LIN {X 0,Y 412.15,Z 242.134,A -85,B 0,C 180,E1 -10569.119,E2 -10569.119} C_VEL
LIN {X 0,Y 411.731,Z 238.226,A -85,B 0,C 180,E1 -10571.737,E2 -10571.737} C_VEL
LIN {X 0,Y 411.199,Z 234.89,A -85,B 0,C 180,E1 -10574.123,E2 -10574.123} C_VEL
LIN {X 0,Y 411.182,Z 234.895,A -85,B 0,C 180,E1 -10577.304,E2 -10577.304} C_VEL
LIN {X 0,Y 411.215,Z 234.89,A -85,B 0,C 180,E1 -10580.776,E2 -10580.776} C_VEL
LIN {X 0,Y 411.198,Z 234.894,A -85,B 0,C 180,E1 -10584.471,E2 -10584.471} C_VEL
LIN {X 0,Y 411.208,Z 234.889,A -85,B 0,C 180,E1 -10586.873,E2 -10586.873} C_VEL
LIN {X 0,Y 411.212,Z 234.891,A -85,B 0,C 180,E1 -10590.65,E2 -10590.65} C_VEL
LIN {X 0,Y 411.195,Z 234.89,A -85,B 0,C 180,E1 -10593.616,E2 -10593.616} C_VEL
LIN {X 0,Y 411.196,Z 234.89,A -85,B 0,C 180,E1 -10596.852,E2 -10596.852} C_VEL
LIN {X 0,Y 411.216,Z 234.887,A -85,B 0,C 180,E1 -10600.051,E2 -10600.051} C_VEL
LIN {X 0,Y 411.264,Z 234.879,A -85,B 0,C 180,E1 -10603.131,E2 -10603.131} C_VEL
LIN {X 0,Y 411.307,Z 234.877,A -85,B 0,C 180,E1 -10606.896,E2 -10606.896} C_VEL
LIN {X 0,Y 411.29,Z 234.876,A -85,B 0,C 180,E1 -10610.161,E2 -10610.161} C_VEL
LIN {X 0,Y 411.394,Z 234.865,A -85,B 0,C 180,E1 -10613.132,E2 -10613.132} C_VEL
LIN {X 0,Y 411.303,Z 234.878,A -85,B 0,C 180,E1 -10615.099,E2 -10615.099} C_VEL
LIN {X 0,Y 411.513,Z 234.851,A -85,B 0,C 180,E1 -10618.043,E2 -10618.043} C_VEL
LIN {X 0,Y 411.635,Z 234.837,A -85,B 0,C 180,E1 -10620,E2 -10620} C_VEL
LIN {X 0,Y 411.449,Z 234.859,A -85,B 0,C 180,E1 -10622.937,E2 -10622.937} C_VEL
LIN {X 0,Y 411.448,Z 234.857,A -85,B 0,C 180,E1 -10626.672,E2 -10626.672} C_VEL
LIN {X 0,Y 411.294,Z 234.88,A -85,B 0,C 180,E1 -10629.839,E2 -10629.839} C_VEL
LIN {X 0,Y 411.307,Z 234.877,A -85,B 0,C 180,E1 -10633.104,E2 -10633.104} C_VEL
LIN {X 0,Y 411.259,Z 234.881,A -85,B 0,C 180,E1 -10636.889,E2 -10636.889} C_VEL
LIN {X 0,Y 411.232,Z 234.884,A -85,B 0,C 180,E1 -10639.987,E2 -10639.987} C_VEL
LIN {X 0,Y 411.197,Z 234.889,A -85,B 0,C 180,E1 -10643.148,E2 -10643.148} C_VEL
LIN {X 0,Y 411.238,Z 234.884,A -85,B 0,C 180,E1 -10646.381,E2 -10646.381} C_VEL
LIN {X 0,Y 411.202,Z 234.888,A -85,B 0,C 180,E1 -10649.713,E2 -10649.713} C_VEL
LIN {X 0,Y 411.208,Z 234.887,A -85,B 0,C 180,E1 -10653.156,E2 -10653.156} C_VEL
LIN {X 0,Y 411.194,Z 234.889,A -85,B 0,C 180,E1 -10656.553,E2 -10656.553} C_VEL
LIN {X 0,Y 411.179,Z 234.89,A -85,B 0,C 180,E1 -10659.722,E2 -10659.722} C_VEL
LIN {X 0,Y 411.166,Z 234.895,A -85,B 0,C 180,E1 -10663.135,E2 -10663.135} C_VEL
LIN {X 0,Y 411.169,Z 234.895,A -85,B 0,C 180,E1 -10665.881,E2 -10665.881} C_VEL
LIN {X 0,Y 411.159,Z 234.898,A -85,B 0,C 180,E1 -10668.773,E2 -10668.773} C_VEL
LIN {X 0,Y 411.159,Z 234.896,A -85,B 0,C 180,E1 -10669.493,E2 -10669.493} C_VEL
LIN {X 0,Y 411.277,Z 236.124,A -85,B 0,C 180,E1 -10670.782,E2 -10670.782} C_VEL
LIN {X 0,Y 411.294,Z 239.248,A -85,B 0,C 180,E1 -10673.429,E2 -10673.429} C_VEL
LIN {X 0,Y 411.162,Z 241.979,A -85,B 0,C 180,E1 -10675.662,E2 -10675.662} C_VEL
LIN {X 0,Y 410.925,Z 246.363,A -85,B 0,C 180,E1 -10679.13,E2 -10679.13} C_VEL
LIN {X 0,Y 410.666,Z 250.766,A -85,B 0,C 180,E1 -10682.479,E2 -10682.479} C_VEL
LIN {X 0,Y 410.562,Z 255.215,A -85,B 0,C 180,E1 -10685.743,E2 -10685.743} C_VEL
LIN {X 0,Y 410.436,Z 259.421,A -85,B 0,C 180,E1 -10688.752,E2 -10688.752} C_VEL
LIN {X 0,Y 414.52,Z 274.317,A -85,B 0,C 180,E1 -10689.4,E2 -10689.4} C_VEL
LIN {X 0,Y 417.537,Z 287.727,A -85,B 0,C 180,E1 -10690.136,E2 -10690.136} C_VEL
LIN {X 0,Y 417.676,Z 291.393,A -85,B 0,C 180,E1 -10690.335,E2 -10690.335} C_VEL
LIN {X 0,Y 416.878,Z 304.123,A -85,B 0,C 180,E1 -10691.091,E2 -10691.091} C_VEL
LIN {X 0,Y 415.949,Z 316.643,A -85,B 0,C 180,E1 -10692.04,E2 -10692.04} C_VEL
LIN {X 0,Y 414.909,Z 328.342,A -85,B 0,C 180,E1 -10693.138,E2 -10693.138} C_VEL
LIN {X 0,Y 413.823,Z 340.015,A -85,B 0,C 180,E1 -10694.485,E2 -10694.485} C_VEL
LIN {X 0,Y 412.756,Z 350.606,A -85,B 0,C 180,E1 -10695.983,E2 -10695.983} C_VEL
LIN {X 0,Y 412.086,Z 359.036,A -85,B 0,C 180,E1 -10697.441,E2 -10697.441} C_VEL
LIN {X 0,Y 411.263,Z 367.277,A -85,B 0,C 180,E1 -10699.165,E2 -10699.165} C_VEL
LIN {X 0,Y 410.811,Z 373.015,A -85,B 0,C 180,E1 -10700.647,E2 -10700.647} C_VEL
LIN {X 0,Y 410.452,Z 377.734,A -85,B 0,C 180,E1 -10702.127,E2 -10702.127} C_VEL
LIN {X 0,Y 410.322,Z 381.154,A -85,B 0,C 180,E1 -10703.428,E2 -10703.428} C_VEL
LIN {X 0,Y 410.101,Z 384.499,A -85,B 0,C 180,E1 -10705.085,E2 -10705.085} C_VEL
LIN {X 0,Y 409.972,Z 387.2,A -85,B 0,C 180,E1 -10707.052,E2 -10707.052} C_VEL
LIN {X 0,Y 409.918,Z 388.555,A -85,B 0,C 180,E1 -10709.018,E2 -10709.018} C_VEL
LIN {X 0,Y 409.918,Z 388.591,A -85,B 0,C 180,E1 -10710.982,E2 -10710.982} C_VEL
LIN {X 0,Y 409.971,Z 387.304,A -85,B 0,C 180,E1 -10712.948,E2 -10712.948} C_VEL
LIN {X 0,Y 410.095,Z 384.665,A -85,B 0,C 180,E1 -10714.916,E2 -10714.916} C_VEL
LIN {X 0,Y 410.321,Z 380.607,A -85,B 0,C 180,E1 -10716.886,E2 -10716.886} C_VEL
LIN {X 0,Y 410.591,Z 375.976,A -85,B 0,C 180,E1 -10718.557,E2 -10718.557} C_VEL
LIN {X 0,Y 410.123,Z 373.603,A -85,B 0,C 180,E1 -10719.305,E2 -10719.305} C_VEL
LIN {X 0,Y 407.665,Z 369.385,A -85,B 0,C 180,E1 -10720.516,E2 -10720.516} C_VEL
LIN {X 0,Y 405.273,Z 364.741,A -85,B 0,C 180,E1 -10721.704,E2 -10721.704} C_VEL
LIN {X 0,Y 404.912,Z 361.52,A -85,B 0,C 180,E1 -10722.406,E2 -10722.406} C_VEL
LIN {X 0,Y 405.639,Z 352.68,A -85,B 0,C 180,E1 -10724.038,E2 -10724.038} C_VEL
LIN {X 0,Y 406.716,Z 342.744,A -85,B 0,C 180,E1 -10725.536,E2 -10725.536} C_VEL
LIN {X 0,Y 407.811,Z 331.683,A -85,B 0,C 180,E1 -10726.907,E2 -10726.907} C_VEL
LIN {X 0,Y 409.011,Z 319.268,A -85,B 0,C 180,E1 -10728.146,E2 -10728.146} C_VEL
LIN {X 0,Y 409.999,Z 307.073,A -85,B 0,C 180,E1 -10729.129,E2 -10729.129} C_VEL
LIN {X 0,Y 410.827,Z 294.562,A -85,B 0,C 180,E1 -10729.931,E2 -10729.931} C_VEL
LIN {X 0,Y 411.06,Z 290.348,A -85,B 0,C 180,E1 -10730.162,E2 -10730.162} C_VEL
LIN {X 0,Y 408.229,Z 277.162,A -85,B 0,C 180,E1 -10730.932,E2 -10730.932} C_VEL
LIN {X 0,Y 404.44,Z 263.529,A -85,B 0,C 180,E1 -10731.585,E2 -10731.585} C_VEL
LIN {X 0,Y 403.377,Z 259.517,A -85,B 0,C 180,E1 -10731.764,E2 -10731.764} C_VEL
LIN {X 0,Y 403.543,Z 254.954,A -85,B 0,C 180,E1 -10735.093,E2 -10735.093} C_VEL
LIN {X 0,Y 403.639,Z 251.022,A -85,B 0,C 180,E1 -10738.042,E2 -10738.042} C_VEL
LIN {X 0,Y 403.826,Z 248.062,A -85,B 0,C 180,E1 -10740.312,E2 -10740.312} C_VEL
LIN {X 0,Y 404.083,Z 243.693,A -85,B 0,C 180,E1 -10743.818,E2 -10743.818} C_VEL
LIN {X 0,Y 404.248,Z 239.971,A -85,B 0,C 180,E1 -10746.896,E2 -10746.896} C_VEL
LIN {X 0,Y 404.171,Z 236.332,A -85,B 0,C 180,E1 -10750.045,E2 -10750.045} C_VEL
LIN {X 0,Y 404.119,Z 235.775,A -85,B 0,C 180,E1 -10751.599,E2 -10751.599} C_VEL
LIN {X 0,Y 404.148,Z 235.771,A -85,B 0,C 180,E1 -10754.522,E2 -10754.522} C_VEL
LIN {X 0,Y 404.127,Z 235.772,A -85,B 0,C 180,E1 -10757.294,E2 -10757.294} C_VEL
LIN {X 0,Y 404.134,Z 235.77,A -85,B 0,C 180,E1 -10759.951,E2 -10759.951} C_VEL
LIN {X 0,Y 404.138,Z 235.77,A -85,B 0,C 180,E1 -10763.125,E2 -10763.125} C_VEL
LIN {X 0,Y 404.147,Z 235.77,A -85,B 0,C 180,E1 -10766.188,E2 -10766.188} C_VEL
LIN {X 0,Y 404.148,Z 235.768,A -85,B 0,C 180,E1 -10769.715,E2 -10769.715} C_VEL
LIN {X 0,Y 404.198,Z 235.761,A -85,B 0,C 180,E1 -10773.123,E2 -10773.123} C_VEL
LIN {X 0,Y 404.177,Z 235.76,A -85,B 0,C 180,E1 -10775.334,E2 -10775.334} C_VEL
LIN {X 0,Y 404.141,Z 235.768,A -85,B 0,C 180,E1 -10778.581,E2 -10778.581} C_VEL
LIN {X 0,Y 404.211,Z 235.759,A -85,B 0,C 180,E1 -10781.762,E2 -10781.762} C_VEL
LIN {X 0,Y 404.209,Z 235.759,A -85,B 0,C 180,E1 -10784.882,E2 -10784.882} C_VEL
LIN {X 0,Y 404.259,Z 235.753,A -85,B 0,C 180,E1 -10787.958,E2 -10787.958} C_VEL
LIN {X 0,Y 404.269,Z 235.751,A -85,B 0,C 180,E1 -10790.998,E2 -10790.998} C_VEL
LIN {X 0,Y 404.417,Z 235.733,A -85,B 0,C 180,E1 -10794.015,E2 -10794.015} C_VEL
LIN {X 0,Y 404.48,Z 235.725,A -85,B 0,C 180,E1 -10798.008,E2 -10798.008} C_VEL
LIN {X 0,Y 404.42,Z 235.733,A -85,B 0,C 180,E1 -10800.996,E2 -10800.996} C_VEL
LIN {X 0,Y 404.418,Z 235.733,A -85,B 0,C 180,E1 -10802.988,E2 -10802.988} C_VEL
LIN {X 0,Y 404.384,Z 235.738,A -85,B 0,C 180,E1 -10805.985,E2 -10805.985} C_VEL
LIN {X 0,Y 404.267,Z 235.752,A -85,B 0,C 180,E1 -10809.001,E2 -10809.001} C_VEL
LIN {X 0,Y 404.259,Z 235.752,A -85,B 0,C 180,E1 -10812.041,E2 -10812.041} C_VEL
LIN {X 0,Y 404.21,Z 235.761,A -85,B 0,C 180,E1 -10815.118,E2 -10815.118} C_VEL
LIN {X 0,Y 404.206,Z 235.761,A -85,B 0,C 180,E1 -10818.238,E2 -10818.238} C_VEL
LIN {X 0,Y 404.141,Z 235.77,A -85,B 0,C 180,E1 -10821.419,E2 -10821.419} C_VEL
LIN {X 0,Y 404.163,Z 235.764,A -85,B 0,C 180,E1 -10824.667,E2 -10824.667} C_VEL
LIN {X 0,Y 404.118,Z 235.771,A -85,B 0,C 180,E1 -10828.005,E2 -10828.005} C_VEL
LIN {X 0,Y 404.146,Z 235.768,A -85,B 0,C 180,E1 -10830.285,E2 -10830.285} C_VEL
LIN {X 0,Y 404.147,Z 235.769,A -85,B 0,C 180,E1 -10833.812,E2 -10833.812} C_VEL
LIN {X 0,Y 404.137,Z 235.772,A -85,B 0,C 180,E1 -10836.875,E2 -10836.875} C_VEL
LIN {X 0,Y 404.149,Z 235.769,A -85,B 0,C 180,E1 -10840.08,E2 -10840.08} C_VEL
LIN {X 0,Y 404.155,Z 235.772,A -85,B 0,C 180,E1 -10843.084,E2 -10843.084} C_VEL
LIN {X 0,Y 404.162,Z 235.921,A -85,B 0,C 180,E1 -10845.71,E2 -10845.71} C_VEL
LIN {X 0,Y 404.829,Z 240.125,A -85,B 0,C 180,E1 -10848.723,E2 -10848.723} C_VEL
LIN {X 0,Y 405.166,Z 244.034,A -85,B 0,C 180,E1 -10851.358,E2 -10851.358} C_VEL
LIN {X 0,Y 404.996,Z 247.953,A -85,B 0,C 180,E1 -10853.842,E2 -10853.842} C_VEL
LIN {X 0,Y 404.579,Z 253.839,A -85,B 0,C 180,E1 -10857.418,E2 -10857.418} C_VEL
LIN {X 0,Y 404.232,Z 259.74,A -85,B 0,C 180,E1 -10860.869,E2 -10860.869} C_VEL
LIN {X 0,Y 404.002,Z 263.62,A -85,B 0,C 180,E1 -10863.109,E2 -10863.109} C_VEL
LIN {X 0,Y 403.608,Z 269.448,A -85,B 0,C 180,E1 -10866.391,E2 -10866.391} C_VEL
LIN {X 0,Y 403.506,Z 272.965,A -85,B 0,C 180,E1 -10868.3,E2 -10868.3} C_VEL
LIN {X 0,Y 407.021,Z 287.509,A -85,B 0,C 180,E1 -10868.898,E2 -10868.898} C_VEL
LIN {X 0,Y 409.374,Z 299.361,A -85,B 0,C 180,E1 -10869.512,E2 -10869.512} C_VEL
LIN {X 0,Y 410.559,Z 307.1,A -85,B 0,C 180,E1 -10869.979,E2 -10869.979} C_VEL
LIN {X 0,Y 409.743,Z 319.944,A -85,B 0,C 180,E1 -10870.769,E2 -10870.769} C_VEL
LIN {X 0,Y 408.695,Z 332.088,A -85,B 0,C 180,E1 -10871.71,E2 -10871.71} C_VEL
LIN {X 0,Y 407.583,Z 343.741,A -85,B 0,C 180,E1 -10872.825,E2 -10872.825} C_VEL
LIN {X 0,Y 406.637,Z 353.442,A -85,B 0,C 180,E1 -10873.947,E2 -10873.947} C_VEL
LIN {X 0,Y 405.605,Z 364.193,A -85,B 0,C 180,E1 -10875.449,E2 -10875.449} C_VEL
LIN {X 0,Y 404.793,Z 373.072,A -85,B 0,C 180,E1 -10876.955,E2 -10876.955} C_VEL
LIN {X 0,Y 404.165,Z 380.463,A -85,B 0,C 180,E1 -10878.464,E2 -10878.464} C_VEL
LIN {X 0,Y 403.632,Z 386.625,A -85,B 0,C 180,E1 -10879.972,E2 -10879.972} C_VEL
LIN {X 0,Y 403.159,Z 393.171,A -85,B 0,C 180,E1 -10881.983,E2 -10881.983} C_VEL
LIN {X 0,Y 402.966,Z 398.072,A -85,B 0,C 180,E1 -10883.993,E2 -10883.993} C_VEL
LIN {X 0,Y 402.827,Z 401.479,A -85,B 0,C 180,E1 -10885.998,E2 -10885.998} C_VEL
LIN {X 0,Y 402.834,Z 403.496,A -85,B 0,C 180,E1 -10888,E2 -10888} C_VEL
LIN {X 0,Y 402.83,Z 404.163,A -85,B 0,C 180,E1 -10890,E2 -10890} C_VEL
LIN {X 0,Y 402.834,Z 403.493,A -85,B 0,C 180,E1 -10892,E2 -10892} C_VEL
LIN {X 0,Y 402.827,Z 401.476,A -85,B 0,C 180,E1 -10894.002,E2 -10894.002} C_VEL
LIN {X 0,Y 402.937,Z 398.063,A -85,B 0,C 180,E1 -10896.007,E2 -10896.007} C_VEL
LIN {X 0,Y 403.093,Z 394.554,A -85,B 0,C 180,E1 -10897.514,E2 -10897.514} C_VEL
LIN {X 0,Y 403.355,Z 390.094,A -85,B 0,C 180,E1 -10899.022,E2 -10899.022} C_VEL
LIN {X 0,Y 403.813,Z 383.66,A -85,B 0,C 180,E1 -10900.783,E2 -10900.783} C_VEL
LIN {X 0,Y 404.59,Z 375.671,A -85,B 0,C 180,E1 -10902.541,E2 -10902.541} C_VEL
LIN {X 0,Y 405.323,Z 367.312,A -85,B 0,C 180,E1 -10904.049,E2 -10904.049} C_VEL
LIN {X 0,Y 406.271,Z 357.251,A -85,B 0,C 180,E1 -10905.553,E2 -10905.553} C_VEL
LIN {X 0,Y 407.365,Z 346.031,A -85,B 0,C 180,E1 -10906.926,E2 -10906.926} C_VEL
LIN {X 0,Y 408.421,Z 334.87,A -85,B 0,C 180,E1 -10908.043,E2 -10908.043} C_VEL
LIN {X 0,Y 409.55,Z 322.718,A -85,B 0,C 180,E1 -10909.029,E2 -10909.029} C_VEL
LIN {X 0,Y 410.375,Z 310.48,A -85,B 0,C 180,E1 -10909.828,E2 -10909.828} C_VEL
LIN {X 0,Y 410.418,Z 305.829,A -85,B 0,C 180,E1 -10910.093,E2 -10910.093} C_VEL
LIN {X 0,Y 407.874,Z 291.298,A -85,B 0,C 180,E1 -10910.911,E2 -10910.911} C_VEL
LIN {X 0,Y 404.428,Z 276.916,A -85,B 0,C 180,E1 -10911.552,E2 -10911.552} C_VEL
LIN {X 0,Y 403.506,Z 272.844,A -85,B 0,C 180,E1 -10911.723,E2 -10911.723} C_VEL
LIN {X 0,Y 403.79,Z 266.654,A -85,B 0,C 180,E1 -10915.168,E2 -10915.168} C_VEL
LIN {X 0,Y 404.12,Z 261.659,A -85,B 0,C 180,E1 -10918.005,E2 -10918.005} C_VEL
LIN {X 0,Y 404.499,Z 255.404,A -85,B 0,C 180,E1 -10921.641,E2 -10921.641} C_VEL
LIN {X 0,Y 404.904,Z 249.255,A -85,B 0,C 180,E1 -10925.335,E2 -10925.335} C_VEL
LIN {X 0,Y 405.121,Z 245.958,A -85,B 0,C 180,E1 -10927.386,E2 -10927.386} C_VEL
LIN {X 0,Y 405.069,Z 242.048,A -85,B 0,C 180,E1 -10929.938,E2 -10929.938} C_VEL
LIN {X 0,Y 404.552,Z 238.144,A -85,B 0,C 180,E1 -10932.65,E2 -10932.65} C_VEL
LIN {X 0,Y 404.156,Z 235.768,A -85,B 0,C 180,E1 -10934.524,E2 -10934.524} C_VEL
LIN {X 0,Y 404.137,Z 235.772,A -85,B 0,C 180,E1 -10937.296,E2 -10937.296} C_VEL
LIN {X 0,Y 404.17,Z 235.767,A -85,B 0,C 180,E1 -10939.955,E2 -10939.955} C_VEL
LIN {X 0,Y 404.136,Z 235.772,A -85,B 0,C 180,E1 -10943.125,E2 -10943.125} C_VEL
LIN {X 0,Y 404.146,Z 235.771,A -85,B 0,C 180,E1 -10946.188,E2 -10946.188} C_VEL
LIN {X 0,Y 404.145,Z 235.768,A -85,B 0,C 180,E1 -10949.715,E2 -10949.715} C_VEL
LIN {X 0,Y 404.135,Z 235.768,A -85,B 0,C 180,E1 -10953.119,E2 -10953.119} C_VEL
LIN {X 0,Y 404.161,Z 235.766,A -85,B 0,C 180,E1 -10956.425,E2 -10956.425} C_VEL
LIN {X 0,Y 404.192,Z 235.761,A -85,B 0,C 180,E1 -10959.874,E2 -10959.874} C_VEL
LIN {X 0,Y 404.217,Z 235.757,A -85,B 0,C 180,E1 -10962.993,E2 -10962.993} C_VEL
LIN {X 0,Y 404.284,Z 235.752,A -85,B 0,C 180,E1 -10966.939,E2 -10966.939} C_VEL
LIN {X 0,Y 404.256,Z 235.751,A -85,B 0,C 180,E1 -10969.988,E2 -10969.988} C_VEL
LIN {X 0,Y 404.344,Z 235.742,A -85,B 0,C 180,E1 -10973.012,E2 -10973.012} C_VEL
LIN {X 0,Y 404.274,Z 235.753,A -85,B 0,C 180,E1 -10975.014,E2 -10975.014} C_VEL
LIN {X 0,Y 404.482,Z 235.726,A -85,B 0,C 180,E1 -10978.009,E2 -10978.009} C_VEL
LIN {X 0,Y 404.605,Z 235.713,A -85,B 0,C 180,E1 -10980,E2 -10980} C_VEL
LIN {X 0,Y 404.408,Z 235.736,A -85,B 0,C 180,E1 -10982.989,E2 -10982.989} C_VEL
LIN {X 0,Y 404.394,Z 235.735,A -85,B 0,C 180,E1 -10986.673,E2 -10986.673} C_VEL
LIN {X 0,Y 404.293,Z 235.748,A -85,B 0,C 180,E1 -10989.001,E2 -10989.001} C_VEL
LIN {X 0,Y 404.258,Z 235.753,A -85,B 0,C 180,E1 -10992.042,E2 -10992.042} C_VEL
LIN {X 0,Y 404.207,Z 235.76,A -85,B 0,C 180,E1 -10995.118,E2 -10995.118} C_VEL
LIN {X 0,Y 404.212,Z 235.76,A -85,B 0,C 180,E1 -10998.238,E2 -10998.238} C_VEL
LIN {X 0,Y 404.14,Z 235.768,A -85,B 0,C 180,E1 -11001.419,E2 -11001.419} C_VEL
LIN {X 0,Y 404.176,Z 235.764,A -85,B 0,C 180,E1 -11004.666,E2 -11004.666} C_VEL
LIN {X 0,Y 404.197,Z 235.761,A -85,B 0,C 180,E1 -11008,E2 -11008} C_VEL
LIN {X 0,Y 404.14,Z 235.767,A -85,B 0,C 180,E1 -11011.558,E2 -11011.558} C_VEL
LIN {X 0,Y 404.185,Z 235.763,A -85,B 0,C 180,E1 -11015.016,E2 -11015.016} C_VEL
LIN {X 0,Y 404.138,Z 235.771,A -85,B 0,C 180,E1 -11018.759,E2 -11018.759} C_VEL
LIN {X 0,Y 404.111,Z 235.773,A -85,B 0,C 180,E1 -11021.598,E2 -11021.598} C_VEL
LIN {X 0,Y 404.145,Z 235.768,A -85,B 0,C 180,E1 -11024.522,E2 -11024.522} C_VEL
LIN {X 0,Y 404.136,Z 235.772,A -85,B 0,C 180,E1 -11027.295,E2 -11027.295} C_VEL
LIN {X 0,Y 404.114,Z 235.776,A -85,B 0,C 180,E1 -11028.634,E2 -11028.634} C_VEL
LIN {X 0,Y 404.17,Z 236.204,A -85,B 0,C 180,E1 -11029.955,E2 -11029.955} C_VEL
LIN {X 0,Y 404.262,Z 239.158,A -85,B 0,C 180,E1 -11032.521,E2 -11032.521} C_VEL
LIN {X 0,Y 404.197,Z 242.084,A -85,B 0,C 180,E1 -11034.985,E2 -11034.985} C_VEL
LIN {X 0,Y 403.905,Z 246.472,A -85,B 0,C 180,E1 -11038.533,E2 -11038.533} C_VEL
LIN {X 0,Y 403.63,Z 250.889,A -85,B 0,C 180,E1 -11041.958,E2 -11041.958} C_VEL
LIN {X 0,Y 403.549,Z 255.337,A -85,B 0,C 180,E1 -11045.293,E2 -11045.293} C_VEL
LIN {X 0,Y 403.372,Z 259.555,A -85,B 0,C 180,E1 -11048.362,E2 -11048.362} C_VEL
LIN {X 0,Y 407.364,Z 273.874,A -85,B 0,C 180,E1 -11048.999,E2 -11048.999} C_VEL
LIN {X 0,Y 410.596,Z 287.877,A -85,B 0,C 180,E1 -11049.785,E2 -11049.785} C_VEL
LIN {X 0,Y 411,Z 291.536,A -85,B 0,C 180,E1 -11050.002,E2 -11050.002} C_VEL
LIN {X 0,Y 410.201,Z 303.521,A -85,B 0,C 180,E1 -11050.716,E2 -11050.716} C_VEL
LIN {X 0,Y 409.349,Z 315.361,A -85,B 0,C 180,E1 -11051.611,E2 -11051.611} C_VEL
LIN {X 0,Y 408.182,Z 327.312,A -85,B 0,C 180,E1 -11052.722,E2 -11052.722} C_VEL
LIN {X 0,Y 407.18,Z 338.209,A -85,B 0,C 180,E1 -11053.969,E2 -11053.969} C_VEL
LIN {X 0,Y 406.224,Z 347.338,A -85,B 0,C 180,E1 -11055.215,E2 -11055.215} C_VEL
LIN {X 0,Y 405.332,Z 356.718,A -85,B 0,C 180,E1 -11056.764,E2 -11056.764} C_VEL
LIN {X 0,Y 404.467,Z 365.205,A -85,B 0,C 180,E1 -11058.473,E2 -11058.473} C_VEL
LIN {X 0,Y 403.913,Z 371.353,A -85,B 0,C 180,E1 -11059.98,E2 -11059.98} C_VEL
LIN {X 0,Y 403.4,Z 377.87,A -85,B 0,C 180,E1 -11061.988,E2 -11061.988} C_VEL
LIN {X 0,Y 403.14,Z 382.755,A -85,B 0,C 180,E1 -11063.996,E2 -11063.996} C_VEL
LIN {X 0,Y 402.89,Z 386.158,A -85,B 0,C 180,E1 -11065.999,E2 -11065.999} C_VEL
LIN {X 0,Y 402.886,Z 388.177,A -85,B 0,C 180,E1 -11068.001,E2 -11068.001} C_VEL
LIN {X 0,Y 402.831,Z 388.872,A -85,B 0,C 180,E1 -11070,E2 -11070} C_VEL
LIN {X 0,Y 402.885,Z 388.247,A -85,B 0,C 180,E1 -11071.999,E2 -11071.999} C_VEL
LIN {X 0,Y 402.888,Z 386.292,A -85,B 0,C 180,E1 -11074.001,E2 -11074.001} C_VEL
LIN {X 0,Y 403.119,Z 382.954,A -85,B 0,C 180,E1 -11076.004,E2 -11076.004} C_VEL
LIN {X 0,Y 403.396,Z 378.141,A -85,B 0,C 180,E1 -11078.012,E2 -11078.012} C_VEL
LIN {X 0,Y 403.894,Z 371.695,A -85,B 0,C 180,E1 -11080.021,E2 -11080.021} C_VEL
LIN {X 0,Y 404.538,Z 364.514,A -85,B 0,C 180,E1 -11081.779,E2 -11081.779} C_VEL
LIN {X 0,Y 404.912,Z 361.52,A -85,B 0,C 180,E1 -11082.406,E2 -11082.406} C_VEL
LIN {X 0,Y 404.444,Z 359.326,A -85,B 0,C 180,E1 -11082.873,E2 -11082.873} C_VEL
LIN {X 0,Y 401.95,Z 355.894,A -85,B 0,C 180,E1 -11083.622,E2 -11083.622} C_VEL
LIN {X 0,Y 399.498,Z 352.264,A -85,B 0,C 180,E1 -11084.357,E2 -11084.357} C_VEL
LIN {X 0,Y 399.096,Z 349.71,A -85,B 0,C 180,E1 -11084.793,E2 -11084.793} C_VEL
LIN {X 0,Y 400.277,Z 339.073,A -85,B 0,C 180,E1 -11086.316,E2 -11086.316} C_VEL
LIN {X 0,Y 401.337,Z 328.321,A -85,B 0,C 180,E1 -11087.582,E2 -11087.582} C_VEL
LIN {X 0,Y 402.514,Z 316.553,A -85,B 0,C 180,E1 -11088.713,E2 -11088.713} C_VEL
LIN {X 0,Y 403.509,Z 303.888,A -85,B 0,C 180,E1 -11089.698,E2 -11089.698} C_VEL
LIN {X 0,Y 404.278,Z 291.107,A -85,B 0,C 180,E1 -11090.478,E2 -11090.478} C_VEL
LIN {X 0,Y 401.163,Z 277.017,A -85,B 0,C 180,E1 -11091.33,E2 -11091.33} C_VEL
LIN {X 0,Y 397.295,Z 263.245,A -85,B 0,C 180,E1 -11092.003,E2 -11092.003} C_VEL
LIN {X 0,Y 396.329,Z 259.667,A -85,B 0,C 180,E1 -11092.158,E2 -11092.158} C_VEL
LIN {X 0,Y 396.504,Z 255.427,A -85,B 0,C 180,E1 -11095.315,E2 -11095.315} C_VEL
LIN {X 0,Y 396.644,Z 251.145,A -85,B 0,C 180,E1 -11098.581,E2 -11098.581} C_VEL
LIN {X 0,Y 396.904,Z 246.717,A -85,B 0,C 180,E1 -11102.088,E2 -11102.088} C_VEL
LIN {X 0,Y 397.179,Z 242.571,A -85,B 0,C 180,E1 -11105.515,E2 -11105.515} C_VEL
LIN {X 0,Y 397.215,Z 239.363,A -85,B 0,C 180,E1 -11108.262,E2 -11108.262} C_VEL
LIN {X 0,Y 397.081,Z 236.935,A -85,B 0,C 180,E1 -11110.442,E2 -11110.442} C_VEL
LIN {X 0,Y 397.064,Z 236.652,A -85,B 0,C 180,E1 -11111.978,E2 -11111.978} C_VEL
LIN {X 0,Y 397.089,Z 236.65,A -85,B 0,C 180,E1 -11115.069,E2 -11115.069} C_VEL
LIN {X 0,Y 397.056,Z 236.654,A -85,B 0,C 180,E1 -11118.023,E2 -11118.023} C_VEL
LIN {X 0,Y 397.096,Z 236.646,A -85,B 0,C 180,E1 -11121.724,E2 -11121.724} C_VEL
LIN {X 0,Y 397.127,Z 236.642,A -85,B 0,C 180,E1 -11125.507,E2 -11125.507} C_VEL
LIN {X 0,Y 397.081,Z 236.651,A -85,B 0,C 180,E1 -11129.118,E2 -11129.118} C_VEL
LIN {X 0,Y 397.197,Z 236.636,A -85,B 0,C 180,E1 -11132.61,E2 -11132.61} C_VEL
LIN {X 0,Y 397.131,Z 236.643,A -85,B 0,C 180,E1 -11135.982,E2 -11135.982} C_VEL
LIN {X 0,Y 397.142,Z 236.638,A -85,B 0,C 180,E1 -11139.705,E2 -11139.705} C_VEL
LIN {X 0,Y 397.185,Z 236.634,A -85,B 0,C 180,E1 -11142.845,E2 -11142.845} C_VEL
LIN {X 0,Y 397.232,Z 236.629,A -85,B 0,C 180,E1 -11146.703,E2 -11146.703} C_VEL
LIN {X 0,Y 397.219,Z 236.629,A -85,B 0,C 180,E1 -11149.809,E2 -11149.809} C_VEL
LIN {X 0,Y 397.337,Z 236.615,A -85,B 0,C 180,E1 -11152.888,E2 -11152.888} C_VEL
LIN {X 0,Y 397.252,Z 236.626,A -85,B 0,C 180,E1 -11154.925,E2 -11154.925} C_VEL
LIN {X 0,Y 397.449,Z 236.601,A -85,B 0,C 180,E1 -11157.973,E2 -11157.973} C_VEL
LIN {X 0,Y 397.384,Z 236.609,A -85,B 0,C 180,E1 -11161.013,E2 -11161.013} C_VEL
LIN {X 0,Y 397.377,Z 236.611,A -85,B 0,C 180,E1 -11163.041,E2 -11163.041} C_VEL
LIN {X 0,Y 397.335,Z 236.616,A -85,B 0,C 180,E1 -11166.092,E2 -11166.092} C_VEL
LIN {X 0,Y 397.237,Z 236.628,A -85,B 0,C 180,E1 -11169.162,E2 -11169.162} C_VEL
LIN {X 0,Y 397.222,Z 236.628,A -85,B 0,C 180,E1 -11172.258,E2 -11172.258} C_VEL
LIN {X 0,Y 397.182,Z 236.635,A -85,B 0,C 180,E1 -11175.392,E2 -11175.392} C_VEL
LIN {X 0,Y 397.159,Z 236.637,A -85,B 0,C 180,E1 -11178.574,E2 -11178.574} C_VEL
LIN {X 0,Y 397.098,Z 236.645,A -85,B 0,C 180,E1 -11181.818,E2 -11181.818} C_VEL
LIN {X 0,Y 397.108,Z 236.641,A -85,B 0,C 180,E1 -11185.135,E2 -11185.135} C_VEL
LIN {X 0,Y 397.071,Z 236.648,A -85,B 0,C 180,E1 -11188.548,E2 -11188.548} C_VEL
LIN {X 0,Y 397.084,Z 236.646,A -85,B 0,C 180,E1 -11191.836,E2 -11191.836} C_VEL
LIN {X 0,Y 397.127,Z 236.645,A -85,B 0,C 180,E1 -11194.493,E2 -11194.493} C_VEL
LIN {X 0,Y 397.103,Z 236.647,A -85,B 0,C 180,E1 -11198.275,E2 -11198.275} C_VEL
LIN {X 0,Y 397.09,Z 236.65,A -85,B 0,C 180,E1 -11200.909,E2 -11200.909} C_VEL
LIN {X 0,Y 397.103,Z 236.652,A -85,B 0,C 180,E1 -11203.648,E2 -11203.648} C_VEL
LIN {X 0,Y 397.133,Z 236.806,A -85,B 0,C 180,E1 -11205.422,E2 -11205.422} C_VEL
LIN {X 0,Y 397.685,Z 240.198,A -85,B 0,C 180,E1 -11207.922,E2 -11207.922} C_VEL
LIN {X 0,Y 398.14,Z 244.562,A -85,B 0,C 180,E1 -11210.959,E2 -11210.959} C_VEL
LIN {X 0,Y 398.057,Z 247.855,A -85,B 0,C 180,E1 -11213.109,E2 -11213.109} C_VEL
LIN {X 0,Y 397.693,Z 252.728,A -85,B 0,C 180,E1 -11216.158,E2 -11216.158} C_VEL
LIN {X 0,Y 397.379,Z 257.671,A -85,B 0,C 180,E1 -11219.143,E2 -11219.143} C_VEL
LIN {X 0,Y 397.025,Z 263.505,A -85,B 0,C 180,E1 -11222.597,E2 -11222.597} C_VEL
LIN {X 0,Y 396.59,Z 269.323,A -85,B 0,C 180,E1 -11225.947,E2 -11225.947} C_VEL
LIN {X 0,Y 396.441,Z 272.81,A -85,B 0,C 180,E1 -11227.892,E2 -11227.892} C_VEL
LIN {X 0,Y 400.109,Z 287.627,A -85,B 0,C 180,E1 -11228.525,E2 -11228.525} C_VEL
LIN {X 0,Y 402.644,Z 300.487,A -85,B 0,C 180,E1 -11229.219,E2 -11229.219} C_VEL
LIN {X 0,Y 403.823,Z 308.952,A -85,B 0,C 180,E1 -11229.747,E2 -11229.747} C_VEL
LIN {X 0,Y 402.932,Z 320.904,A -85,B 0,C 180,E1 -11230.513,E2 -11230.513} C_VEL
LIN {X 0,Y 401.808,Z 333.385,A -85,B 0,C 180,E1 -11231.517,E2 -11231.517} C_VEL
LIN {X 0,Y 400.642,Z 344.785,A -85,B 0,C 180,E1 -11232.65,E2 -11232.65} C_VEL
LIN {X 0,Y 399.588,Z 355.265,A -85,B 0,C 180,E1 -11233.918,E2 -11233.918} C_VEL
LIN {X 0,Y 398.556,Z 365.692,A -85,B 0,C 180,E1 -11235.447,E2 -11235.447} C_VEL
LIN {X 0,Y 397.69,Z 374.297,A -85,B 0,C 180,E1 -11236.978,E2 -11236.978} C_VEL
LIN {X 0,Y 396.909,Z 382.537,A -85,B 0,C 180,E1 -11238.768,E2 -11238.768} C_VEL
LIN {X 0,Y 396.447,Z 388.308,A -85,B 0,C 180,E1 -11240.304,E2 -11240.304} C_VEL
LIN {X 0,Y 396.093,Z 393.036,A -85,B 0,C 180,E1 -11241.839,E2 -11241.839} C_VEL
LIN {X 0,Y 395.889,Z 397.938,A -85,B 0,C 180,E1 -11243.885,E2 -11243.885} C_VEL
LIN {X 0,Y 395.75,Z 401.345,A -85,B 0,C 180,E1 -11245.926,E2 -11245.926} C_VEL
LIN {X 0,Y 395.731,Z 403.361,A -85,B 0,C 180,E1 -11247.964,E2 -11247.964} C_VEL
LIN {X 0,Y 395.758,Z 404.029,A -85,B 0,C 180,E1 -11250,E2 -11250} C_VEL
LIN {X 0,Y 395.731,Z 403.358,A -85,B 0,C 180,E1 -11252.035,E2 -11252.035} C_VEL
LIN {X 0,Y 395.75,Z 401.34,A -85,B 0,C 180,E1 -11254.073,E2 -11254.073} C_VEL
LIN {X 0,Y 395.859,Z 397.819,A -85,B 0,C 180,E1 -11256.167,E2 -11256.167} C_VEL
LIN {X 0,Y 396.092,Z 393.017,A -85,B 0,C 180,E1 -11258.16,E2 -11258.16} C_VEL
LIN {X 0,Y 396.572,Z 386.466,A -85,B 0,C 180,E1 -11260.208,E2 -11260.208} C_VEL
LIN {X 0,Y 397.259,Z 379.18,A -85,B 0,C 180,E1 -11261.998,E2 -11261.998} C_VEL
LIN {X 0,Y 398.036,Z 371.016,A -85,B 0,C 180,E1 -11263.631,E2 -11263.631} C_VEL
LIN {X 0,Y 398.867,Z 362.383,A -85,B 0,C 180,E1 -11265.064,E2 -11265.064} C_VEL
LIN {X 0,Y 399.995,Z 351.277,A -85,B 0,C 180,E1 -11266.59,E2 -11266.59} C_VEL
LIN {X 0,Y 401.134,Z 339.94,A -85,B 0,C 180,E1 -11267.855,E2 -11267.855} C_VEL
LIN {X 0,Y 402.364,Z 327.407,A -85,B 0,C 180,E1 -11268.985,E2 -11268.985} C_VEL
LIN {X 0,Y 403.443,Z 314.089,A -85,B 0,C 180,E1 -11269.938,E2 -11269.938} C_VEL
LIN {X 0,Y 403.81,Z 308.747,A -85,B 0,C 180,E1 -11270.257,E2 -11270.257} C_VEL
LIN {X 0,Y 401.834,Z 295.997,A -85,B 0,C 180,E1 -11271.03,E2 -11271.03} C_VEL
LIN {X 0,Y 398.792,Z 282.188,A -85,B 0,C 180,E1 -11271.721,E2 -11271.721} C_VEL
LIN {X 0,Y 396.428,Z 272.711,A -85,B 0,C 180,E1 -11272.13,E2 -11272.13} C_VEL
LIN {X 0,Y 396.738,Z 266.965,A -85,B 0,C 180,E1 -11275.386,E2 -11275.386} C_VEL
LIN {X 0,Y 397.105,Z 261.536,A -85,B 0,C 180,E1 -11278.545,E2 -11278.545} C_VEL
LIN {X 0,Y 397.482,Z 255.677,A -85,B 0,C 180,E1 -11282.035,E2 -11282.035} C_VEL
LIN {X 0,Y 397.926,Z 249.751,A -85,B 0,C 180,E1 -11285.666,E2 -11285.666} C_VEL
LIN {X 0,Y 398.117,Z 245.862,A -85,B 0,C 180,E1 -11288.16,E2 -11288.16} C_VEL
LIN {X 0,Y 397.936,Z 242.276,A -85,B 0,C 180,E1 -11290.586,E2 -11290.586} C_VEL
LIN {X 0,Y 397.333,Z 238.063,A -85,B 0,C 180,E1 -11293.617,E2 -11293.617} C_VEL
LIN {X 0,Y 397.114,Z 236.647,A -85,B 0,C 180,E1 -11294.755,E2 -11294.755} C_VEL
LIN {X 0,Y 397.067,Z 236.652,A -85,B 0,C 180,E1 -11298.021,E2 -11298.021} C_VEL
LIN {X 0,Y 397.129,Z 236.646,A -85,B 0,C 180,E1 -11301.139,E2 -11301.139} C_VEL
LIN {X 0,Y 397.12,Z 236.647,A -85,B 0,C 180,E1 -11304.497,E2 -11304.497} C_VEL
LIN {X 0,Y 397.079,Z 236.65,A -85,B 0,C 180,E1 -11307.929,E2 -11307.929} C_VEL
LIN {X 0,Y 397.118,Z 236.643,A -85,B 0,C 180,E1 -11310.295,E2 -11310.295} C_VEL
LIN {X 0,Y 397.095,Z 236.647,A -85,B 0,C 180,E1 -11313.739,E2 -11313.739} C_VEL
LIN {X 0,Y 397.105,Z 236.647,A -85,B 0,C 180,E1 -11317.085,E2 -11317.085} C_VEL
LIN {X 0,Y 397.147,Z 236.642,A -85,B 0,C 180,E1 -11320.353,E2 -11320.353} C_VEL
LIN {X 0,Y 397.168,Z 236.638,A -85,B 0,C 180,E1 -11323.553,E2 -11323.553} C_VEL
LIN {X 0,Y 397.23,Z 236.628,A -85,B 0,C 180,E1 -11326.703,E2 -11326.703} C_VEL
LIN {X 0,Y 397.217,Z 236.626,A -85,B 0,C 180,E1 -11329.809,E2 -11329.809} C_VEL
LIN {X 0,Y 397.296,Z 236.619,A -85,B 0,C 180,E1 -11332.887,E2 -11332.887} C_VEL
LIN {X 0,Y 397.244,Z 236.629,A -85,B 0,C 180,E1 -11334.925,E2 -11334.925} C_VEL
LIN {X 0,Y 397.451,Z 236.602,A -85,B 0,C 180,E1 -11337.973,E2 -11337.973} C_VEL
LIN {X 0,Y 397.574,Z 236.589,A -85,B 0,C 180,E1 -11340,E2 -11340} C_VEL
LIN {X 0,Y 397.367,Z 236.614,A -85,B 0,C 180,E1 -11343.042,E2 -11343.042} C_VEL
LIN {X 0,Y 397.345,Z 236.613,A -85,B 0,C 180,E1 -11346.671,E2 -11346.671} C_VEL
LIN {X 0,Y 397.254,Z 236.625,A -85,B 0,C 180,E1 -11349.162,E2 -11349.162} C_VEL
LIN {X 0,Y 397.221,Z 236.629,A -85,B 0,C 180,E1 -11352.258,E2 -11352.258} C_VEL
LIN {X 0,Y 397.18,Z 236.634,A -85,B 0,C 180,E1 -11355.392,E2 -11355.392} C_VEL
LIN {X 0,Y 397.164,Z 236.636,A -85,B 0,C 180,E1 -11358.573,E2 -11358.573} C_VEL
LIN {X 0,Y 397.098,Z 236.644,A -85,B 0,C 180,E1 -11361.819,E2 -11361.819} C_VEL
LIN {X 0,Y 397.154,Z 236.639,A -85,B 0,C 180,E1 -11365.512,E2 -11365.512} C_VEL
LIN {X 0,Y 397.123,Z 236.641,A -85,B 0,C 180,E1 -11368.544,E2 -11368.544} C_VEL
LIN {X 0,Y 397.08,Z 236.649,A -85,B 0,C 180,E1 -11372.072,E2 -11372.072} C_VEL
LIN {X 0,Y 397.12,Z 236.645,A -85,B 0,C 180,E1 -11375.503,E2 -11375.503} C_VEL
LIN {X 0,Y 397.096,Z 236.649,A -85,B 0,C 180,E1 -11378.855,E2 -11378.855} C_VEL
LIN {X 0,Y 397.058,Z 236.655,A -85,B 0,C 180,E1 -11382.269,E2 -11382.269} C_VEL
LIN {X 0,Y 397.088,Z 236.649,A -85,B 0,C 180,E1 -11385.069,E2 -11385.069} C_VEL
LIN {X 0,Y 397.064,Z 236.653,A -85,B 0,C 180,E1 -11388.022,E2 -11388.022} C_VEL
LIN {X 0,Y 397.082,Z 236.818,A -85,B 0,C 180,E1 -11389.558,E2 -11389.558} C_VEL
LIN {X 0,Y 397.241,Z 239.248,A -85,B 0,C 180,E1 -11391.741,E2 -11391.741} C_VEL
LIN {X 0,Y 397.179,Z 242.436,A -85,B 0,C 180,E1 -11394.485,E2 -11394.485} C_VEL
LIN {X 0,Y 396.901,Z 246.938,A -85,B 0,C 180,E1 -11398.206,E2 -11398.206} C_VEL
LIN {X 0,Y 396.629,Z 251.012,A -85,B 0,C 180,E1 -11401.418,E2 -11401.418} C_VEL
LIN {X 0,Y 396.481,Z 255.477,A -85,B 0,C 180,E1 -11404.823,E2 -11404.823} C_VEL
LIN {X 0,Y 396.339,Z 259.829,A -85,B 0,C 180,E1 -11407.963,E2 -11407.963} C_VEL
LIN {X 0,Y 400.506,Z 274.377,A -85,B 0,C 180,E1 -11408.635,E2 -11408.635} C_VEL
LIN {X 0,Y 403.641,Z 287.934,A -85,B 0,C 180,E1 -11409.417,E2 -11409.417} C_VEL
LIN {X 0,Y 404.336,Z 291.679,A -85,B 0,C 180,E1 -11409.658,E2 -11409.658} C_VEL
LIN {X 0,Y 403.482,Z 304.022,A -85,B 0,C 180,E1 -11410.409,E2 -11410.409} C_VEL
LIN {X 0,Y 402.458,Z 316.923,A -85,B 0,C 180,E1 -11411.416,E2 -11411.416} C_VEL
LIN {X 0,Y 401.274,Z 328.622,A -85,B 0,C 180,E1 -11412.547,E2 -11412.547} C_VEL
LIN {X 0,Y 400.132,Z 340.293,A -85,B 0,C 180,E1 -11413.94,E2 -11413.94} C_VEL
LIN {X 0,Y 398.983,Z 350.718,A -85,B 0,C 180,E1 -11415.463,E2 -11415.463} C_VEL
LIN {X 0,Y 398.172,Z 359.312,A -85,B 0,C 180,E1 -11416.994,E2 -11416.994} C_VEL
LIN {X 0,Y 397.244,Z 367.552,A -85,B 0,C 180,E1 -11418.778,E2 -11418.778} C_VEL
LIN {X 0,Y 396.729,Z 373.289,A -85,B 0,C 180,E1 -11420.312,E2 -11420.312} C_VEL
LIN {X 0,Y 396.366,Z 378.006,A -85,B 0,C 180,E1 -11421.845,E2 -11421.845} C_VEL
LIN {X 0,Y 396.067,Z 382.891,A -85,B 0,C 180,E1 -11423.888,E2 -11423.888} C_VEL
LIN {X 0,Y 395.815,Z 386.293,A -85,B 0,C 180,E1 -11425.927,E2 -11425.927} C_VEL
LIN {X 0,Y 395.786,Z 388.312,A -85,B 0,C 180,E1 -11427.965,E2 -11427.965} C_VEL
LIN {X 0,Y 395.759,Z 389.006,A -85,B 0,C 180,E1 -11430,E2 -11430} C_VEL
LIN {X 0,Y 395.785,Z 388.382,A -85,B 0,C 180,E1 -11432.035,E2 -11432.035} C_VEL
LIN {X 0,Y 395.813,Z 386.426,A -85,B 0,C 180,E1 -11434.073,E2 -11434.073} C_VEL
LIN {X 0,Y 396.057,Z 383.088,A -85,B 0,C 180,E1 -11436.112,E2 -11436.112} C_VEL
LIN {X 0,Y 396.362,Z 378.275,A -85,B 0,C 180,E1 -11438.155,E2 -11438.155} C_VEL
LIN {X 0,Y 396.884,Z 371.828,A -85,B 0,C 180,E1 -11440.2,E2 -11440.2} C_VEL
LIN {X 0,Y 397.583,Z 364.647,A -85,B 0,C 180,E1 -11441.988,E2 -11441.988} C_VEL
LIN {X 0,Y 398.394,Z 356.823,A -85,B 0,C 180,E1 -11443.575,E2 -11443.575} C_VEL
LIN {X 0,Y 399.096,Z 349.71,A -85,B 0,C 180,E1 -11444.793,E2 -11444.793} C_VEL
LIN {X 0,Y 398.861,Z 345.783,A -85,B 0,C 180,E1 -11445.423,E2 -11445.423} C_VEL
LIN {X 0,Y 396.756,Z 339.219,A -85,B 0,C 180,E1 -11446.454,E2 -11446.454} C_VEL
LIN {X 0,Y 394.763,Z 332.301,A -85,B 0,C 180,E1 -11447.438,E2 -11447.438} C_VEL
LIN {X 0,Y 394.677,Z 327.682,A -85,B 0,C 180,E1 -11447.977,E2 -11447.977} C_VEL
LIN {X 0,Y 395.926,Z 315.258,A -85,B 0,C 180,E1 -11449.171,E2 -11449.171} C_VEL
LIN {X 0,Y 396.968,Z 302.216,A -85,B 0,C 180,E1 -11450.168,E2 -11450.168} C_VEL
LIN {X 0,Y 397.582,Z 292.36,A -85,B 0,C 180,E1 -11450.772,E2 -11450.772} C_VEL
LIN {X 0,Y 394.405,Z 277.903,A -85,B 0,C 180,E1 -11451.682,E2 -11451.682} C_VEL
LIN {X 0,Y 390.311,Z 263.539,A -85,B 0,C 180,E1 -11452.414,E2 -11452.414} C_VEL
LIN {X 0,Y 389.309,Z 259.792,A -85,B 0,C 180,E1 -11452.594,E2 -11452.594} C_VEL
LIN {X 0,Y 389.441,Z 255.741,A -85,B 0,C 180,E1 -11455.665,E2 -11455.665} C_VEL
LIN {X 0,Y 389.637,Z 251.257,A -85,B 0,C 180,E1 -11459.144,E2 -11459.144} C_VEL
LIN {X 0,Y 389.891,Z 246.826,A -85,B 0,C 180,E1 -11462.736,E2 -11462.736} C_VEL
LIN {X 0,Y 390.143,Z 243.13,A -85,B 0,C 180,E1 -11465.843,E2 -11465.843} C_VEL
LIN {X 0,Y 390.149,Z 239.448,A -85,B 0,C 180,E1 -11469.086,E2 -11469.086} C_VEL
LIN {X 0,Y 390.019,Z 237.582,A -85,B 0,C 180,E1 -11470.815,E2 -11470.815} C_VEL
LIN {X 0,Y 390.057,Z 237.525,A -85,B 0,C 180,E1 -11473.886,E2 -11473.886} C_VEL
LIN {X 0,Y 390.054,Z 237.526,A -85,B 0,C 180,E1 -11476.789,E2 -11476.789} C_VEL
LIN {X 0,Y 390.013,Z 237.53,A -85,B 0,C 180,E1 -11479.555,E2 -11479.555} C_VEL
LIN {X 0,Y 390.043,Z 237.525,A -85,B 0,C 180,E1 -11482.45,E2 -11482.45} C_VEL
LIN {X 0,Y 390.071,Z 237.524,A -85,B 0,C 180,E1 -11485.975,E2 -11485.975} C_VEL
LIN {X 0,Y 390.049,Z 237.524,A -85,B 0,C 180,E1 -11489.869,E2 -11489.869} C_VEL
LIN {X 0,Y 390.116,Z 237.515,A -85,B 0,C 180,E1 -11493.232,E2 -11493.232} C_VEL
LIN {X 0,Y 390.07,Z 237.521,A -85,B 0,C 180,E1 -11496.764,E2 -11496.764} C_VEL
LIN {X 0,Y 390.107,Z 237.515,A -85,B 0,C 180,E1 -11499.983,E2 -11499.983} C_VEL
LIN {X 0,Y 390.141,Z 237.512,A -85,B 0,C 180,E1 -11503.248,E2 -11503.248} C_VEL
LIN {X 0,Y 390.198,Z 237.504,A -85,B 0,C 180,E1 -11506.562,E2 -11506.562} C_VEL
LIN {X 0,Y 390.17,Z 237.507,A -85,B 0,C 180,E1 -11509.623,E2 -11509.623} C_VEL
LIN {X 0,Y 390.285,Z 237.493,A -85,B 0,C 180,E1 -11512.758,E2 -11512.758} C_VEL
LIN {X 0,Y 390.224,Z 237.501,A -85,B 0,C 180,E1 -11514.833,E2 -11514.833} C_VEL
LIN {X 0,Y 390.418,Z 237.477,A -85,B 0,C 180,E1 -11517.937,E2 -11517.937} C_VEL
LIN {X 0,Y 390.349,Z 237.486,A -85,B 0,C 180,E1 -11521.032,E2 -11521.032} C_VEL
LIN {X 0,Y 390.311,Z 237.491,A -85,B 0,C 180,E1 -11523.096,E2 -11523.096} C_VEL
LIN {X 0,Y 390.288,Z 237.495,A -85,B 0,C 180,E1 -11526.202,E2 -11526.202} C_VEL
LIN {X 0,Y 390.195,Z 237.506,A -85,B 0,C 180,E1 -11529.329,E2 -11529.329} C_VEL
LIN {X 0,Y 390.174,Z 237.507,A -85,B 0,C 180,E1 -11532.483,E2 -11532.483} C_VEL
LIN {X 0,Y 390.142,Z 237.512,A -85,B 0,C 180,E1 -11535.677,E2 -11535.677} C_VEL
LIN {X 0,Y 390.104,Z 237.516,A -85,B 0,C 180,E1 -11538.922,E2 -11538.922} C_VEL
LIN {X 0,Y 390.04,Z 237.525,A -85,B 0,C 180,E1 -11542.234,E2 -11542.234} C_VEL
LIN {X 0,Y 390.051,Z 237.521,A -85,B 0,C 180,E1 -11545.722,E2 -11545.722} C_VEL
LIN {X 0,Y 390.03,Z 237.529,A -85,B 0,C 180,E1 -11549.112,E2 -11549.112} C_VEL
LIN {X 0,Y 390.045,Z 237.526,A -85,B 0,C 180,E1 -11552.721,E2 -11552.721} C_VEL
LIN {X 0,Y 390.057,Z 237.528,A -85,B 0,C 180,E1 -11555.825,E2 -11555.825} C_VEL
LIN {X 0,Y 390.07,Z 237.524,A -85,B 0,C 180,E1 -11559.218,E2 -11559.218} C_VEL
LIN {X 0,Y 390.045,Z 237.531,A -85,B 0,C 180,E1 -11562.374,E2 -11562.374} C_VEL
LIN {X 0,Y 390.053,Z 237.559,A -85,B 0,C 180,E1 -11565.014,E2 -11565.014} C_VEL
LIN {X 0,Y 390.746,Z 241.907,A -85,B 0,C 180,E1 -11568.28,E2 -11568.28} C_VEL
LIN {X 0,Y 391.134,Z 245.812,A -85,B 0,C 180,E1 -11571.032,E2 -11571.032} C_VEL
LIN {X 0,Y 390.917,Z 250.322,A -85,B 0,C 180,E1 -11574,E2 -11574} C_VEL
LIN {X 0,Y 390.517,Z 255.601,A -85,B 0,C 180,E1 -11577.323,E2 -11577.323} C_VEL
LIN {X 0,Y 390.105,Z 261.444,A -85,B 0,C 180,E1 -11580.894,E2 -11580.894} C_VEL
LIN {X 0,Y 389.698,Z 267.255,A -85,B 0,C 180,E1 -11584.353,E2 -11584.353} C_VEL
LIN {X 0,Y 389.41,Z 272.607,A -85,B 0,C 180,E1 -11587.463,E2 -11587.463} C_VEL
LIN {X 0,Y 393.443,Z 288.825,A -85,B 0,C 180,E1 -11588.193,E2 -11588.193} C_VEL
LIN {X 0,Y 395.906,Z 301.448,A -85,B 0,C 180,E1 -11588.905,E2 -11588.905} C_VEL
LIN {X 0,Y 397.079,Z 310.385,A -85,B 0,C 180,E1 -11589.481,E2 -11589.481} C_VEL
LIN {X 0,Y 396.081,Z 322.549,A -85,B 0,C 180,E1 -11590.298,E2 -11590.298} C_VEL
LIN {X 0,Y 394.912,Z 334.679,A -85,B 0,C 180,E1 -11591.317,E2 -11591.317} C_VEL
LIN {X 0,Y 393.635,Z 346.922,A -85,B 0,C 180,E1 -11592.599,E2 -11592.599} C_VEL
LIN {X 0,Y 392.537,Z 357.03,A -85,B 0,C 180,E1 -11593.888,E2 -11593.888} C_VEL
LIN {X 0,Y 391.472,Z 367.081,A -85,B 0,C 180,E1 -11595.443,E2 -11595.443} C_VEL
LIN {X 0,Y 390.596,Z 375.431,A -85,B 0,C 180,E1 -11597.002,E2 -11597.002} C_VEL
LIN {X 0,Y 389.929,Z 382.403,A -85,B 0,C 180,E1 -11598.565,E2 -11598.565} C_VEL
LIN {X 0,Y 389.396,Z 388.173,A -85,B 0,C 180,E1 -11600.127,E2 -11600.127} C_VEL
LIN {X 0,Y 389.042,Z 392.902,A -85,B 0,C 180,E1 -11601.69,E2 -11601.69} C_VEL
LIN {X 0,Y 388.799,Z 397.803,A -85,B 0,C 180,E1 -11603.773,E2 -11603.773} C_VEL
LIN {X 0,Y 388.675,Z 401.211,A -85,B 0,C 180,E1 -11605.852,E2 -11605.852} C_VEL
LIN {X 0,Y 388.628,Z 403.226,A -85,B 0,C 180,E1 -11607.927,E2 -11607.927} C_VEL
LIN {X 0,Y 388.671,Z 403.894,A -85,B 0,C 180,E1 -11610,E2 -11610} C_VEL
LIN {X 0,Y 388.628,Z 403.223,A -85,B 0,C 180,E1 -11612.073,E2 -11612.073} C_VEL
LIN {X 0,Y 388.674,Z 401.205,A -85,B 0,C 180,E1 -11614.148,E2 -11614.148} C_VEL
LIN {X 0,Y 388.793,Z 397.792,A -85,B 0,C 180,E1 -11616.226,E2 -11616.226} C_VEL
LIN {X 0,Y 389.042,Z 392.881,A -85,B 0,C 180,E1 -11618.309,E2 -11618.309} C_VEL
LIN {X 0,Y 389.396,Z 388.147,A -85,B 0,C 180,E1 -11619.873,E2 -11619.873} C_VEL
LIN {X 0,Y 390.062,Z 381.284,A -85,B 0,C 180,E1 -11621.695,E2 -11621.695} C_VEL
LIN {X 0,Y 390.897,Z 372.765,A -85,B 0,C 180,E1 -11623.517,E2 -11623.517} C_VEL
LIN {X 0,Y 391.79,Z 363.877,A -85,B 0,C 180,E1 -11625.076,E2 -11625.076} C_VEL
LIN {X 0,Y 392.923,Z 353.115,A -85,B 0,C 180,E1 -11626.63,E2 -11626.63} C_VEL
LIN {X 0,Y 394.095,Z 342.226,A -85,B 0,C 180,E1 -11627.916,E2 -11627.916} C_VEL
LIN {X 0,Y 395.335,Z 330.309,A -85,B 0,C 180,E1 -11629.066,E2 -11629.066} C_VEL
LIN {X 0,Y 396.492,Z 317.72,A -85,B 0,C 180,E1 -11630.041,E2 -11630.041} C_VEL
LIN {X 0,Y 397.008,Z 308.772,A -85,B 0,C 180,E1 -11630.61,E2 -11630.61} C_VEL
LIN {X 0,Y 394.611,Z 294.338,A -85,B 0,C 180,E1 -11631.502,E2 -11631.502} C_VEL
LIN {X 0,Y 391.269,Z 279.82,A -85,B 0,C 180,E1 -11632.227,E2 -11632.227} C_VEL
LIN {X 0,Y 389.393,Z 272.619,A -85,B 0,C 180,E1 -11632.521,E2 -11632.521} C_VEL
LIN {X 0,Y 389.697,Z 267.235,A -85,B 0,C 180,E1 -11635.647,E2 -11635.647} C_VEL
LIN {X 0,Y 390.015,Z 263.257,A -85,B 0,C 180,E1 -11637.997,E2 -11637.997} C_VEL
LIN {X 0,Y 390.356,Z 257.535,A -85,B 0,C 180,E1 -11641.474,E2 -11641.474} C_VEL
LIN {X 0,Y 390.789,Z 251.644,A -85,B 0,C 180,E1 -11645.134,E2 -11645.134} C_VEL
LIN {X 0,Y 391.093,Z 247.595,A -85,B 0,C 180,E1 -11647.75,E2 -11647.75} C_VEL
LIN {X 0,Y 391.107,Z 245.133,A -85,B 0,C 180,E1 -11649.404,E2 -11649.404} C_VEL
LIN {X 0,Y 390.587,Z 240.862,A -85,B 0,C 180,E1 -11652.461,E2 -11652.461} C_VEL
LIN {X 0,Y 390.049,Z 237.529,A -85,B 0,C 180,E1 -11654.988,E2 -11654.988} C_VEL
LIN {X 0,Y 390.032,Z 237.529,A -85,B 0,C 180,E1 -11658.187,E2 -11658.187} C_VEL
LIN {X 0,Y 390.089,Z 237.522,A -85,B 0,C 180,E1 -11660.908,E2 -11660.908} C_VEL
LIN {X 0,Y 390.086,Z 237.522,A -85,B 0,C 180,E1 -11664.793,E2 -11664.793} C_VEL
LIN {X 0,Y 390.024,Z 237.528,A -85,B 0,C 180,E1 -11668.496,E2 -11668.496} C_VEL
LIN {X 0,Y 390.038,Z 237.526,A -85,B 0,C 180,E1 -11672.064,E2 -11672.064} C_VEL
LIN {X 0,Y 390.055,Z 237.526,A -85,B 0,C 180,E1 -11675.518,E2 -11675.518} C_VEL
LIN {X 0,Y 390.057,Z 237.526,A -85,B 0,C 180,E1 -11678.878,E2 -11678.878} C_VEL
LIN {X 0,Y 390.112,Z 237.516,A -85,B 0,C 180,E1 -11682.166,E2 -11682.166} C_VEL
LIN {X 0,Y 390.146,Z 237.511,A -85,B 0,C 180,E1 -11685.393,E2 -11685.393} C_VEL
LIN {X 0,Y 390.149,Z 237.511,A -85,B 0,C 180,E1 -11688.571,E2 -11688.571} C_VEL
LIN {X 0,Y 390.258,Z 237.498,A -85,B 0,C 180,E1 -11692.086,E2 -11692.086} C_VEL
LIN {X 0,Y 390.214,Z 237.504,A -85,B 0,C 180,E1 -11694.833,E2 -11694.833} C_VEL
LIN {X 0,Y 390.42,Z 237.477,A -85,B 0,C 180,E1 -11697.937,E2 -11697.937} C_VEL
LIN {X 0,Y 390.544,Z 237.464,A -85,B 0,C 180,E1 -11700,E2 -11700} C_VEL
LIN {X 0,Y 390.302,Z 237.494,A -85,B 0,C 180,E1 -11703.097,E2 -11703.097} C_VEL
LIN {X 0,Y 390.3,Z 237.491,A -85,B 0,C 180,E1 -11706.667,E2 -11706.667} C_VEL
LIN {X 0,Y 390.207,Z 237.504,A -85,B 0,C 180,E1 -11709.329,E2 -11709.329} C_VEL
LIN {X 0,Y 390.196,Z 237.504,A -85,B 0,C 180,E1 -11713.439,E2 -11713.439} C_VEL
LIN {X 0,Y 390.151,Z 237.511,A -85,B 0,C 180,E1 -11717.308,E2 -11717.308} C_VEL
LIN {X 0,Y 390.089,Z 237.517,A -85,B 0,C 180,E1 -11720.47,E2 -11720.47} C_VEL
LIN {X 0,Y 390.079,Z 237.522,A -85,B 0,C 180,E1 -11724.481,E2 -11724.481} C_VEL
LIN {X 0,Y 390.119,Z 237.515,A -85,B 0,C 180,E1 -11727.93,E2 -11727.93} C_VEL
LIN {X 0,Y 390.025,Z 237.526,A -85,B 0,C 180,E1 -11731.504,E2 -11731.504} C_VEL
LIN {X 0,Y 390.086,Z 237.52,A -85,B 0,C 180,E1 -11735.207,E2 -11735.207} C_VEL
LIN {X 0,Y 390.061,Z 237.524,A -85,B 0,C 180,E1 -11739.096,E2 -11739.096} C_VEL
LIN {X 0,Y 390.033,Z 237.53,A -85,B 0,C 180,E1 -11742.373,E2 -11742.373} C_VEL
LIN {X 0,Y 390.045,Z 237.528,A -85,B 0,C 180,E1 -11745.354,E2 -11745.354} C_VEL
LIN {X 0,Y 390.027,Z 237.53,A -85,B 0,C 180,E1 -11748.186,E2 -11748.186} C_VEL
LIN {X 0,Y 390.035,Z 237.528,A -85,B 0,C 180,E1 -11749.183,E2 -11749.183} C_VEL
LIN {X 0,Y 390.182,Z 239.355,A -85,B 0,C 180,E1 -11750.919,E2 -11750.919} C_VEL
LIN {X 0,Y 390.148,Z 243.028,A -85,B 0,C 180,E1 -11754.156,E2 -11754.156} C_VEL
LIN {X 0,Y 389.885,Z 246.689,A -85,B 0,C 180,E1 -11757.264,E2 -11757.264} C_VEL
LIN {X 0,Y 389.629,Z 251.126,A -85,B 0,C 180,E1 -11760.855,E2 -11760.855} C_VEL
LIN {X 0,Y 389.44,Z 255.777,A -85,B 0,C 180,E1 -11764.465,E2 -11764.465} C_VEL
LIN {X 0,Y 389.312,Z 259.872,A -85,B 0,C 180,E1 -11767.541,E2 -11767.541} C_VEL
LIN {X 0,Y 393.238,Z 273.603,A -85,B 0,C 180,E1 -11768.185,E2 -11768.185} C_VEL
LIN {X 0,Y 396.391,Z 286.705,A -85,B 0,C 180,E1 -11768.95,E2 -11768.95} C_VEL
LIN {X 0,Y 397.592,Z 293.187,A -85,B 0,C 180,E1 -11769.379,E2 -11769.379} C_VEL
LIN {X 0,Y 396.677,Z 306.105,A -85,B 0,C 180,E1 -11770.208,E2 -11770.208} C_VEL
LIN {X 0,Y 395.595,Z 318.485,A -85,B 0,C 180,E1 -11771.216,E2 -11771.216} C_VEL
LIN {X 0,Y 394.381,Z 329.931,A -85,B 0,C 180,E1 -11772.365,E2 -11772.365} C_VEL
LIN {X 0,Y 393.288,Z 340.431,A -85,B 0,C 180,E1 -11773.653,E2 -11773.653} C_VEL
LIN {X 0,Y 392.095,Z 350.856,A -85,B 0,C 180,E1 -11775.202,E2 -11775.202} C_VEL
LIN {X 0,Y 391.236,Z 359.449,A -85,B 0,C 180,E1 -11776.76,E2 -11776.76} C_VEL
LIN {X 0,Y 390.253,Z 367.689,A -85,B 0,C 180,E1 -11778.574,E2 -11778.574} C_VEL
LIN {X 0,Y 389.709,Z 373.426,A -85,B 0,C 180,E1 -11780.135,E2 -11780.135} C_VEL
LIN {X 0,Y 389.322,Z 378.143,A -85,B 0,C 180,E1 -11781.697,E2 -11781.697} C_VEL
LIN {X 0,Y 389.011,Z 383.027,A -85,B 0,C 180,E1 -11783.777,E2 -11783.777} C_VEL
LIN {X 0,Y 388.743,Z 386.428,A -85,B 0,C 180,E1 -11785.853,E2 -11785.853} C_VEL
LIN {X 0,Y 388.686,Z 388.447,A -85,B 0,C 180,E1 -11787.928,E2 -11787.928} C_VEL
LIN {X 0,Y 388.671,Z 389.141,A -85,B 0,C 180,E1 -11790,E2 -11790} C_VEL
LIN {X 0,Y 388.685,Z 388.516,A -85,B 0,C 180,E1 -11792.073,E2 -11792.073} C_VEL
LIN {X 0,Y 388.741,Z 386.56,A -85,B 0,C 180,E1 -11794.147,E2 -11794.147} C_VEL
LIN {X 0,Y 388.991,Z 383.222,A -85,B 0,C 180,E1 -11796.223,E2 -11796.223} C_VEL
LIN {X 0,Y 389.318,Z 378.408,A -85,B 0,C 180,E1 -11798.304,E2 -11798.304} C_VEL
LIN {X 0,Y 389.882,Z 371.962,A -85,B 0,C 180,E1 -11800.385,E2 -11800.385} C_VEL
LIN {X 0,Y 390.63,Z 364.78,A -85,B 0,C 180,E1 -11802.205,E2 -11802.205} C_VEL
LIN {X 0,Y 391.431,Z 357.205,A -85,B 0,C 180,E1 -11803.772,E2 -11803.772} C_VEL
LIN {X 0,Y 392.379,Z 348.214,A -85,B 0,C 180,E1 -11805.319,E2 -11805.319} C_VEL
LIN {X 0,Y 393.668,Z 337.257,A -85,B 0,C 180,E1 -11806.864,E2 -11806.864} C_VEL
LIN {X 0,Y 394.677,Z 327.682,A -85,B 0,C 180,E1 -11807.977,E2 -11807.977} C_VEL
LIN {X 0,Y 394.612,Z 322.988,A -85,B 0,C 180,E1 -11808.498,E2 -11808.498} C_VEL
LIN {X 0,Y 392.679,Z 315.267,A -85,B 0,C 180,E1 -11809.361,E2 -11809.361} C_VEL
LIN {X 0,Y 390.615,Z 307.201,A -85,B 0,C 180,E1 -11810.152,E2 -11810.152} C_VEL
LIN {X 0,Y 390.333,Z 301.966,A -85,B 0,C 180,E1 -11810.552,E2 -11810.552} C_VEL
LIN {X 0,Y 390.86,Z 293.613,A -85,B 0,C 180,E1 -11811.077,E2 -11811.077} C_VEL
LIN {X 0,Y 387.804,Z 279.51,A -85,B 0,C 180,E1 -11812.002,E2 -11812.002} C_VEL
LIN {X 0,Y 383.828,Z 265.275,A -85,B 0,C 180,E1 -11812.768,E2 -11812.768} C_VEL
LIN {X 0,Y 382.235,Z 259.925,A -85,B 0,C 180,E1 -11813.036,E2 -11813.036} C_VEL
LIN {X 0,Y 382.387,Z 255.865,A -85,B 0,C 180,E1 -11816.175,E2 -11816.175} C_VEL
LIN {X 0,Y 382.623,Z 251.379,A -85,B 0,C 180,E1 -11819.732,E2 -11819.732} C_VEL
LIN {X 0,Y 382.821,Z 248.15,A -85,B 0,C 180,E1 -11822.382,E2 -11822.382} C_VEL
LIN {X 0,Y 383.018,Z 245.441,A -85,B 0,C 180,E1 -11824.668,E2 -11824.668} C_VEL
LIN {X 0,Y 383.139,Z 241.742,A -85,B 0,C 180,E1 -11827.93,E2 -11827.93} C_VEL
LIN {X 0,Y 383.085,Z 239.565,A -85,B 0,C 180,E1 -11829.949,E2 -11829.949} C_VEL
LIN {X 0,Y 382.965,Z 238.412,A -85,B 0,C 180,E1 -11831.35,E2 -11831.35} C_VEL
LIN {X 0,Y 382.998,Z 238.406,A -85,B 0,C 180,E1 -11834.303,E2 -11834.303} C_VEL
LIN {X 0,Y 383.012,Z 238.403,A -85,B 0,C 180,E1 -11837.24,E2 -11837.24} C_VEL
LIN {X 0,Y 382.989,Z 238.403,A -85,B 0,C 180,E1 -11840.419,E2 -11840.419} C_VEL
LIN {X 0,Y 383.027,Z 238.4,A -85,B 0,C 180,E1 -11844.044,E2 -11844.044} C_VEL
LIN {X 0,Y 382.989,Z 238.406,A -85,B 0,C 180,E1 -11847.578,E2 -11847.578} C_VEL
LIN {X 0,Y 382.995,Z 238.402,A -85,B 0,C 180,E1 -11850.3,E2 -11850.3} C_VEL
LIN {X 0,Y 383.083,Z 238.393,A -85,B 0,C 180,E1 -11854.021,E2 -11854.021} C_VEL
LIN {X 0,Y 382.995,Z 238.405,A -85,B 0,C 180,E1 -11857.334,E2 -11857.334} C_VEL
LIN {X 0,Y 383.063,Z 238.397,A -85,B 0,C 180,E1 -11860.716,E2 -11860.716} C_VEL
LIN {X 0,Y 383.084,Z 238.392,A -85,B 0,C 180,E1 -11864.027,E2 -11864.027} C_VEL
LIN {X 0,Y 383.139,Z 238.387,A -85,B 0,C 180,E1 -11867.284,E2 -11867.284} C_VEL
LIN {X 0,Y 383.146,Z 238.386,A -85,B 0,C 180,E1 -11870.498,E2 -11870.498} C_VEL
LIN {X 0,Y 383.275,Z 238.369,A -85,B 0,C 180,E1 -11873.683,E2 -11873.683} C_VEL
LIN {X 0,Y 383.385,Z 238.352,A -85,B 0,C 180,E1 -11877.899,E2 -11877.899} C_VEL
LIN {X 0,Y 383.315,Z 238.362,A -85,B 0,C 180,E1 -11881.05,E2 -11881.05} C_VEL
LIN {X 0,Y 383.248,Z 238.371,A -85,B 0,C 180,E1 -11883.154,E2 -11883.154} C_VEL
LIN {X 0,Y 383.245,Z 238.373,A -85,B 0,C 180,E1 -11886.317,E2 -11886.317} C_VEL
LIN {X 0,Y 383.145,Z 238.385,A -85,B 0,C 180,E1 -11889.502,E2 -11889.502} C_VEL
LIN {X 0,Y 383.128,Z 238.386,A -85,B 0,C 180,E1 -11893.536,E2 -11893.536} C_VEL
LIN {X 0,Y 383.097,Z 238.389,A -85,B 0,C 180,E1 -11897.069,E2 -11897.069} C_VEL
LIN {X 0,Y 383.031,Z 238.398,A -85,B 0,C 180,E1 -11900.647,E2 -11900.647} C_VEL
LIN {X 0,Y 383.016,Z 238.4,A -85,B 0,C 180,E1 -11903.808,E2 -11903.808} C_VEL
LIN {X 0,Y 382.984,Z 238.404,A -85,B 0,C 180,E1 -11907.307,E2 -11907.307} C_VEL
LIN {X 0,Y 382.984,Z 238.404,A -85,B 0,C 180,E1 -11910.918,E2 -11910.918} C_VEL
LIN {X 0,Y 383.02,Z 238.402,A -85,B 0,C 180,E1 -11914.668,E2 -11914.668} C_VEL
LIN {X 0,Y 383,Z 238.404,A -85,B 0,C 180,E1 -11917.903,E2 -11917.903} C_VEL
LIN {X 0,Y 382.985,Z 238.406,A -85,B 0,C 180,E1 -11921.347,E2 -11921.347} C_VEL
LIN {X 0,Y 383.026,Z 238.524,A -85,B 0,C 180,E1 -11924.764,E2 -11924.764} C_VEL
LIN {X 0,Y 383.558,Z 241.817,A -85,B 0,C 180,E1 -11927.315,E2 -11927.315} C_VEL
LIN {X 0,Y 384.036,Z 245.8,A -85,B 0,C 180,E1 -11930.23,E2 -11930.23} C_VEL
LIN {X 0,Y 383.994,Z 249.621,A -85,B 0,C 180,E1 -11932.844,E2 -11932.844} C_VEL
LIN {X 0,Y 383.686,Z 253.709,A -85,B 0,C 180,E1 -11935.514,E2 -11935.514} C_VEL
LIN {X 0,Y 383.424,Z 257.448,A -85,B 0,C 180,E1 -11937.889,E2 -11937.889} C_VEL
LIN {X 0,Y 383.002,Z 263.264,A -85,B 0,C 180,E1 -11941.504,E2 -11941.504} C_VEL
LIN {X 0,Y 382.525,Z 269.052,A -85,B 0,C 180,E1 -11945.003,E2 -11945.003} C_VEL
LIN {X 0,Y 382.36,Z 272.487,A -85,B 0,C 180,E1 -11947.031,E2 -11947.031} C_VEL
LIN {X 0,Y 386.154,Z 287.42,A -85,B 0,C 180,E1 -11947.71,E2 -11947.71} C_VEL
LIN {X 0,Y 388.97,Z 301.315,A -85,B 0,C 180,E1 -11948.51,E2 -11948.51} C_VEL
LIN {X 0,Y 390.363,Z 311.176,A -85,B 0,C 180,E1 -11949.171,E2 -11949.171} C_VEL
LIN {X 0,Y 389.227,Z 324.067,A -85,B 0,C 180,E1 -11950.073,E2 -11950.073} C_VEL
LIN {X 0,Y 387.879,Z 337.163,A -85,B 0,C 180,E1 -11951.239,E2 -11951.239} C_VEL
LIN {X 0,Y 386.602,Z 348.934,A -85,B 0,C 180,E1 -11952.545,E2 -11952.545} C_VEL
LIN {X 0,Y 385.465,Z 358.683,A -85,B 0,C 180,E1 -11953.856,E2 -11953.856} C_VEL
LIN {X 0,Y 384.419,Z 368.236,A -85,B 0,C 180,E1 -11955.404,E2 -11955.404} C_VEL
LIN {X 0,Y 383.528,Z 376.533,A -85,B 0,C 180,E1 -11957.028,E2 -11957.028} C_VEL
LIN {X 0,Y 382.697,Z 384.293,A -85,B 0,C 180,E1 -11958.882,E2 -11958.882} C_VEL
LIN {X 0,Y 382.219,Z 389.711,A -85,B 0,C 180,E1 -11960.474,E2 -11960.474} C_VEL
LIN {X 0,Y 381.842,Z 395.413,A -85,B 0,C 180,E1 -11962.597,E2 -11962.597} C_VEL
LIN {X 0,Y 381.62,Z 399.551,A -85,B 0,C 180,E1 -11964.717,E2 -11964.717} C_VEL
LIN {X 0,Y 381.509,Z 402.253,A -85,B 0,C 180,E1 -11966.832,E2 -11966.832} C_VEL
LIN {X 0,Y 381.553,Z 403.593,A -85,B 0,C 180,E1 -11968.944,E2 -11968.944} C_VEL
LIN {X 0,Y 381.553,Z 403.591,A -85,B 0,C 180,E1 -11971.055,E2 -11971.055} C_VEL
LIN {X 0,Y 381.509,Z 402.248,A -85,B 0,C 180,E1 -11973.168,E2 -11973.168} C_VEL
LIN {X 0,Y 381.612,Z 399.542,A -85,B 0,C 180,E1 -11975.283,E2 -11975.283} C_VEL
LIN {X 0,Y 381.841,Z 395.395,A -85,B 0,C 180,E1 -11977.402,E2 -11977.402} C_VEL
LIN {X 0,Y 382.218,Z 389.685,A -85,B 0,C 180,E1 -11979.525,E2 -11979.525} C_VEL
LIN {X 0,Y 382.793,Z 383.25,A -85,B 0,C 180,E1 -11981.383,E2 -11981.383} C_VEL
LIN {X 0,Y 383.628,Z 375.258,A -85,B 0,C 180,E1 -11983.238,E2 -11983.238} C_VEL
LIN {X 0,Y 384.562,Z 366.899,A -85,B 0,C 180,E1 -11984.824,E2 -11984.824} C_VEL
LIN {X 0,Y 385.654,Z 356.837,A -85,B 0,C 180,E1 -11986.407,E2 -11986.407} C_VEL
LIN {X 0,Y 386.918,Z 345.615,A -85,B 0,C 180,E1 -11987.849,E2 -11987.849} C_VEL
LIN {X 0,Y 388.17,Z 334.453,A -85,B 0,C 180,E1 -11989.02,E2 -11989.02} C_VEL
LIN {X 0,Y 389.417,Z 322.298,A -85,B 0,C 180,E1 -11990.054,E2 -11990.054} C_VEL
LIN {X 0,Y 390.289,Z 309.935,A -85,B 0,C 180,E1 -11990.902,E2 -11990.902} C_VEL
LIN {X 0,Y 387.94,Z 295.722,A -85,B 0,C 180,E1 -11991.82,E2 -11991.82} C_VEL
LIN {X 0,Y 384.722,Z 281.477,A -85,B 0,C 180,E1 -11992.571,E2 -11992.571} C_VEL
LIN {X 0,Y 382.372,Z 272.43,A -85,B 0,C 180,E1 -11992.991,E2 -11992.991} C_VEL
LIN {X 0,Y 382.68,Z 267.098,A -85,B 0,C 180,E1 -11996.153,E2 -11996.153} C_VEL
LIN {X 0,Y 382.999,Z 263.242,A -85,B 0,C 180,E1 -11998.496,E2 -11998.496} C_VEL
LIN {X 0,Y 383.235,Z 259.37,A -85,B 0,C 180,E1 -12000.896,E2 -12000.896} C_VEL
LIN {X 0,Y 383.531,Z 255.457,A -85,B 0,C 180,E1 -12003.349,E2 -12003.349} C_VEL
LIN {X 0,Y 383.947,Z 250.795,A -85,B 0,C 180,E1 -12006.351,E2 -12006.351} C_VEL
LIN {X 0,Y 384.097,Z 247.625,A -85,B 0,C 180,E1 -12008.471,E2 -12008.471} C_VEL
LIN {X 0,Y 383.798,Z 243.586,A -85,B 0,C 180,E1 -12011.342,E2 -12011.342} C_VEL
LIN {X 0,Y 383.23,Z 239.626,A -85,B 0,C 180,E1 -12014.339,E2 -12014.339} C_VEL
LIN {X 0,Y 383.025,Z 238.405,A -85,B 0,C 180,E1 -12015.419,E2 -12015.419} C_VEL
LIN {X 0,Y 382.989,Z 238.405,A -85,B 0,C 180,E1 -12018.796,E2 -12018.796} C_VEL
LIN {X 0,Y 382.999,Z 238.404,A -85,B 0,C 180,E1 -12022.097,E2 -12022.097} C_VEL
LIN {X 0,Y 383.019,Z 238.402,A -85,B 0,C 180,E1 -12025.332,E2 -12025.332} C_VEL
LIN {X 0,Y 382.983,Z 238.407,A -85,B 0,C 180,E1 -12029.081,E2 -12029.081} C_VEL
LIN {X 0,Y 382.993,Z 238.404,A -85,B 0,C 180,E1 -12032.693,E2 -12032.693} C_VEL
LIN {X 0,Y 383.016,Z 238.4,A -85,B 0,C 180,E1 -12036.192,E2 -12036.192} C_VEL
LIN {X 0,Y 383.057,Z 238.394,A -85,B 0,C 180,E1 -12039.599,E2 -12039.599} C_VEL
LIN {X 0,Y 383.095,Z 238.388,A -85,B 0,C 180,E1 -12042.931,E2 -12042.931} C_VEL
LIN {X 0,Y 383.127,Z 238.383,A -85,B 0,C 180,E1 -12046.464,E2 -12046.464} C_VEL
LIN {X 0,Y 383.131,Z 238.38,A -85,B 0,C 180,E1 -12049.43,E2 -12049.43} C_VEL
LIN {X 0,Y 383.201,Z 238.375,A -85,B 0,C 180,E1 -12052.624,E2 -12052.624} C_VEL
LIN {X 0,Y 383.184,Z 238.379,A -85,B 0,C 180,E1 -12054.738,E2 -12054.738} C_VEL
LIN {X 0,Y 383.387,Z 238.353,A -85,B 0,C 180,E1 -12057.899,E2 -12057.899} C_VEL
LIN {X 0,Y 383.513,Z 238.34,A -85,B 0,C 180,E1 -12060,E2 -12060} C_VEL
LIN {X 0,Y 383.238,Z 238.375,A -85,B 0,C 180,E1 -12063.154,E2 -12063.154} C_VEL
LIN {X 0,Y 383.259,Z 238.369,A -85,B 0,C 180,E1 -12066.66,E2 -12066.66} C_VEL
LIN {X 0,Y 383.153,Z 238.383,A -85,B 0,C 180,E1 -12069.502,E2 -12069.502} C_VEL
LIN {X 0,Y 383.127,Z 238.384,A -85,B 0,C 180,E1 -12073.536,E2 -12073.536} C_VEL
LIN {X 0,Y 383.097,Z 238.39,A -85,B 0,C 180,E1 -12077.455,E2 -12077.455} C_VEL
LIN {X 0,Y 383.03,Z 238.397,A -85,B 0,C 180,E1 -12080.647,E2 -12080.647} C_VEL
LIN {X 0,Y 383.024,Z 238.398,A -85,B 0,C 180,E1 -12083.808,E2 -12083.808} C_VEL
LIN {X 0,Y 383.081,Z 238.393,A -85,B 0,C 180,E1 -12086.123,E2 -12086.123} C_VEL
LIN {X 0,Y 382.994,Z 238.402,A -85,B 0,C 180,E1 -12089.7,E2 -12089.7} C_VEL
LIN {X 0,Y 383.005,Z 238.401,A -85,B 0,C 180,E1 -12093.401,E2 -12093.401} C_VEL
LIN {X 0,Y 383.033,Z 238.398,A -85,B 0,C 180,E1 -12096.164,E2 -12096.164} C_VEL
LIN {X 0,Y 382.977,Z 238.404,A -85,B 0,C 180,E1 -12099.963,E2 -12099.963} C_VEL
LIN {X 0,Y 383.007,Z 238.403,A -85,B 0,C 180,E1 -12102.779,E2 -12102.779} C_VEL
LIN {X 0,Y 382.998,Z 238.404,A -85,B 0,C 180,E1 -12105.789,E2 -12105.789} C_VEL
LIN {X 0,Y 382.974,Z 238.409,A -85,B 0,C 180,E1 -12108.799,E2 -12108.799} C_VEL
LIN {X 0,Y 383.126,Z 239.816,A -85,B 0,C 180,E1 -12110.394,E2 -12110.394} C_VEL
LIN {X 0,Y 383.141,Z 242.397,A -85,B 0,C 180,E1 -12112.748,E2 -12112.748} C_VEL
LIN {X 0,Y 382.994,Z 245.732,A -85,B 0,C 180,E1 -12115.666,E2 -12115.666} C_VEL
LIN {X 0,Y 382.701,Z 249.752,A -85,B 0,C 180,E1 -12119.056,E2 -12119.056} C_VEL
LIN {X 0,Y 382.424,Z 254.233,A -85,B 0,C 180,E1 -12122.649,E2 -12122.649} C_VEL
LIN {X 0,Y 382.33,Z 257.235,A -85,B 0,C 180,E1 -12124.989,E2 -12124.989} C_VEL
LIN {X 0,Y 382.247,Z 260.108,A -85,B 0,C 180,E1 -12127.104,E2 -12127.104} C_VEL
LIN {X 0,Y 386.48,Z 274.537,A -85,B 0,C 180,E1 -12127.813,E2 -12127.813} C_VEL
LIN {X 0,Y 389.617,Z 287.649,A -85,B 0,C 180,E1 -12128.609,E2 -12128.609} C_VEL
LIN {X 0,Y 390.839,Z 294.968,A -85,B 0,C 180,E1 -12129.106,E2 -12129.106} C_VEL
LIN {X 0,Y 389.864,Z 307.827,A -85,B 0,C 180,E1 -12129.97,E2 -12129.97} C_VEL
LIN {X 0,Y 388.7,Z 320.048,A -85,B 0,C 180,E1 -12131.007,E2 -12131.007} C_VEL
LIN {X 0,Y 387.49,Z 331.24,A -85,B 0,C 180,E1 -12132.178,E2 -12132.178} C_VEL
LIN {X 0,Y 386.242,Z 342.489,A -85,B 0,C 180,E1 -12133.618,E2 -12133.618} C_VEL
LIN {X 0,Y 384.998,Z 352.535,A -85,B 0,C 180,E1 -12135.193,E2 -12135.193} C_VEL
LIN {X 0,Y 384.152,Z 360.869,A -85,B 0,C 180,E1 -12136.78,E2 -12136.78} C_VEL
LIN {X 0,Y 383.157,Z 368.832,A -85,B 0,C 180,E1 -12138.628,E2 -12138.628} C_VEL
LIN {X 0,Y 382.549,Z 375.236,A -85,B 0,C 180,E1 -12140.483,E2 -12140.483} C_VEL
LIN {X 0,Y 382.057,Z 380.915,A -85,B 0,C 180,E1 -12142.602,E2 -12142.602} C_VEL
LIN {X 0,Y 381.805,Z 385.041,A -85,B 0,C 180,E1 -12144.719,E2 -12144.719} C_VEL
LIN {X 0,Y 381.589,Z 387.742,A -85,B 0,C 180,E1 -12146.833,E2 -12146.833} C_VEL
LIN {X 0,Y 381.575,Z 389.093,A -85,B 0,C 180,E1 -12148.945,E2 -12148.945} C_VEL
LIN {X 0,Y 381.575,Z 389.128,A -85,B 0,C 180,E1 -12151.055,E2 -12151.055} C_VEL
LIN {X 0,Y 381.587,Z 387.842,A -85,B 0,C 180,E1 -12153.168,E2 -12153.168} C_VEL
LIN {X 0,Y 381.796,Z 385.201,A -85,B 0,C 180,E1 -12155.281,E2 -12155.281} C_VEL
LIN {X 0,Y 382.057,Z 381.143,A -85,B 0,C 180,E1 -12157.398,E2 -12157.398} C_VEL
LIN {X 0,Y 382.522,Z 375.534,A -85,B 0,C 180,E1 -12159.518,E2 -12159.518} C_VEL
LIN {X 0,Y 383.116,Z 369.201,A -85,B 0,C 180,E1 -12161.374,E2 -12161.374} C_VEL
LIN {X 0,Y 384.127,Z 361.319,A -85,B 0,C 180,E1 -12163.221,E2 -12163.221} C_VEL
LIN {X 0,Y 384.953,Z 353.077,A -85,B 0,C 180,E1 -12164.809,E2 -12164.809} C_VEL
LIN {X 0,Y 386.2,Z 343.139,A -85,B 0,C 180,E1 -12166.384,E2 -12166.384} C_VEL
LIN {X 0,Y 387.435,Z 332.076,A -85,B 0,C 180,E1 -12167.825,E2 -12167.825} C_VEL
LIN {X 0,Y 388.627,Z 321.057,A -85,B 0,C 180,E1 -12168.997,E2 -12168.997} C_VEL
LIN {X 0,Y 389.788,Z 309.094,A -85,B 0,C 180,E1 -12170.034,E2 -12170.034} C_VEL
LIN {X 0,Y 390.333,Z 301.966,A -85,B 0,C 180,E1 -12170.552,E2 -12170.552} C_VEL
LIN {X 0,Y 390.175,Z 298.447,A -85,B 0,C 180,E1 -12170.806,E2 -12170.806} C_VEL
LIN {X 0,Y 389.301,Z 295.079,A -85,B 0,C 180,E1 -12171.077,E2 -12171.077} C_VEL
LIN {X 0,Y 386.33,Z 288.738,A -85,B 0,C 180,E1 -12171.635,E2 -12171.635} C_VEL
LIN {X 0,Y 381.081,Z 279.122,A -85,B 0,C 180,E1 -12172.439,E2 -12172.439} C_VEL
LIN {X 0,Y 379.768,Z 275.602,A -85,B 0,C 180,E1 -12172.667,E2 -12172.667} C_VEL
LIN {X 0,Y 375.798,Z 262.561,A -85,B 0,C 180,E1 -12173.359,E2 -12173.359} C_VEL
LIN {X 0,Y 375.188,Z 260.091,A -85,B 0,C 180,E1 -12173.473,E2 -12173.473} C_VEL
LIN {X 0,Y 375.352,Z 255.984,A -85,B 0,C 180,E1 -12176.704,E2 -12176.704} C_VEL
LIN {X 0,Y 375.66,Z 251.162,A -85,B 0,C 180,E1 -12180.617,E2 -12180.617} C_VEL
LIN {X 0,Y 375.978,Z 246.396,A -85,B 0,C 180,E1 -12184.667,E2 -12184.667} C_VEL
LIN {X 0,Y 376.089,Z 244.083,A -85,B 0,C 180,E1 -12186.726,E2 -12186.726} C_VEL
LIN {X 0,Y 376.058,Z 240.577,A -85,B 0,C 180,E1 -12189.983,E2 -12189.983} C_VEL
LIN {X 0,Y 375.961,Z 239.661,A -85,B 0,C 180,E1 -12190.865,E2 -12190.865} C_VEL
LIN {X 0,Y 375.928,Z 239.285,A -85,B 0,C 180,E1 -12192.301,E2 -12192.301} C_VEL
LIN {X 0,Y 375.928,Z 239.285,A -85,B 0,C 180,E1 -12195.269,E2 -12195.269} C_VEL
LIN {X 0,Y 375.92,Z 239.286,A -85,B 0,C 180,E1 -12198.402,E2 -12198.402} C_VEL
LIN {X 0,Y 375.957,Z 239.279,A -85,B 0,C 180,E1 -12201.91,E2 -12201.91} C_VEL
LIN {X 0,Y 375.982,Z 239.276,A -85,B 0,C 180,E1 -12205.333,E2 -12205.333} C_VEL
LIN {X 0,Y 375.96,Z 239.278,A -85,B 0,C 180,E1 -12208.438,E2 -12208.438} C_VEL
LIN {X 0,Y 375.986,Z 239.276,A -85,B 0,C 180,E1 -12212.14,E2 -12212.14} C_VEL
LIN {X 0,Y 376.008,Z 239.269,A -85,B 0,C 180,E1 -12214.539,E2 -12214.539} C_VEL
LIN {X 0,Y 375.96,Z 239.278,A -85,B 0,C 180,E1 -12218.045,E2 -12218.045} C_VEL
LIN {X 0,Y 376.011,Z 239.271,A -85,B 0,C 180,E1 -12221.473,E2 -12221.473} C_VEL
LIN {X 0,Y 376.061,Z 239.265,A -85,B 0,C 180,E1 -12224.833,E2 -12224.833} C_VEL
LIN {X 0,Y 376.052,Z 239.267,A -85,B 0,C 180,E1 -12228.137,E2 -12228.137} C_VEL
LIN {X 0,Y 376.203,Z 239.249,A -85,B 0,C 180,E1 -12231.94,E2 -12231.94} C_VEL
LIN {X 0,Y 376.168,Z 239.251,A -85,B 0,C 180,E1 -12234.64,E2 -12234.64} C_VEL
LIN {X 0,Y 376.351,Z 239.229,A -85,B 0,C 180,E1 -12237.86,E2 -12237.86} C_VEL
LIN {X 0,Y 376.281,Z 239.238,A -85,B 0,C 180,E1 -12241.07,E2 -12241.07} C_VEL
LIN {X 0,Y 376.186,Z 239.252,A -85,B 0,C 180,E1 -12243.213,E2 -12243.213} C_VEL
LIN {X 0,Y 376.203,Z 239.251,A -85,B 0,C 180,E1 -12246.436,E2 -12246.436} C_VEL
LIN {X 0,Y 376.115,Z 239.261,A -85,B 0,C 180,E1 -12249.681,E2 -12249.681} C_VEL
LIN {X 0,Y 376.092,Z 239.262,A -85,B 0,C 180,E1 -12253.658,E2 -12253.658} C_VEL
LIN {X 0,Y 376.035,Z 239.269,A -85,B 0,C 180,E1 -12257.4,E2 -12257.4} C_VEL
LIN {X 0,Y 375.981,Z 239.278,A -85,B 0,C 180,E1 -12260.832,E2 -12260.832} C_VEL
LIN {X 0,Y 375.974,Z 239.279,A -85,B 0,C 180,E1 -12264.283,E2 -12264.283} C_VEL
LIN {X 0,Y 375.928,Z 239.283,A -85,B 0,C 180,E1 -12267.864,E2 -12267.864} C_VEL
LIN {X 0,Y 375.959,Z 239.278,A -85,B 0,C 180,E1 -12271.562,E2 -12271.562} C_VEL
LIN {X 0,Y 375.959,Z 239.283,A -85,B 0,C 180,E1 -12275.415,E2 -12275.415} C_VEL
LIN {X 0,Y 375.975,Z 239.279,A -85,B 0,C 180,E1 -12278.27,E2 -12278.27} C_VEL
LIN {X 0,Y 375.936,Z 239.284,A -85,B 0,C 180,E1 -12281.601,E2 -12281.601} C_VEL
LIN {X 0,Y 376,Z 239.484,A -85,B 0,C 180,E1 -12284.504,E2 -12284.504} C_VEL
LIN {X 0,Y 376.737,Z 244.284,A -85,B 0,C 180,E1 -12288.262,E2 -12288.262} C_VEL
LIN {X 0,Y 377.043,Z 247.576,A -85,B 0,C 180,E1 -12290.672,E2 -12290.672} C_VEL
LIN {X 0,Y 376.949,Z 251.473,A -85,B 0,C 180,E1 -12293.371,E2 -12293.371} C_VEL
LIN {X 0,Y 376.461,Z 257.336,A -85,B 0,C 180,E1 -12297.221,E2 -12297.221} C_VEL
LIN {X 0,Y 375.982,Z 263.132,A -85,B 0,C 180,E1 -12300.922,E2 -12300.922} C_VEL
LIN {X 0,Y 375.518,Z 268.934,A -85,B 0,C 180,E1 -12304.503,E2 -12304.503} C_VEL
LIN {X 0,Y 375.308,Z 272.355,A -85,B 0,C 180,E1 -12306.574,E2 -12306.574} C_VEL
LIN {X 0,Y 379.202,Z 287.129,A -85,B 0,C 180,E1 -12307.273,E2 -12307.273} C_VEL
LIN {X 0,Y 382.073,Z 301.209,A -85,B 0,C 180,E1 -12308.104,E2 -12308.104} C_VEL
LIN {X 0,Y 383.579,Z 311.044,A -85,B 0,C 180,E1 -12308.785,E2 -12308.785} C_VEL
LIN {X 0,Y 382.486,Z 324.562,A -85,B 0,C 180,E1 -12309.762,E2 -12309.762} C_VEL
LIN {X 0,Y 381.148,Z 337.032,A -85,B 0,C 180,E1 -12310.895,E2 -12310.895} C_VEL
LIN {X 0,Y 379.785,Z 348.801,A -85,B 0,C 180,E1 -12312.221,E2 -12312.221} C_VEL
LIN {X 0,Y 378.618,Z 358.55,A -85,B 0,C 180,E1 -12313.556,E2 -12313.556} C_VEL
LIN {X 0,Y 377.474,Z 368.259,A -85,B 0,C 180,E1 -12315.158,E2 -12315.158} C_VEL
LIN {X 0,Y 376.536,Z 376.399,A -85,B 0,C 180,E1 -12316.783,E2 -12316.783} C_VEL
LIN {X 0,Y 375.673,Z 384.158,A -85,B 0,C 180,E1 -12318.672,E2 -12318.672} C_VEL
LIN {X 0,Y 375.167,Z 389.576,A -85,B 0,C 180,E1 -12320.294,E2 -12320.294} C_VEL
LIN {X 0,Y 374.752,Z 395.279,A -85,B 0,C 180,E1 -12322.457,E2 -12322.457} C_VEL
LIN {X 0,Y 374.534,Z 399.417,A -85,B 0,C 180,E1 -12324.616,E2 -12324.616} C_VEL
LIN {X 0,Y 374.426,Z 402.119,A -85,B 0,C 180,E1 -12326.772,E2 -12326.772} C_VEL
LIN {X 0,Y 374.453,Z 403.458,A -85,B 0,C 180,E1 -12328.924,E2 -12328.924} C_VEL
LIN {X 0,Y 374.453,Z 403.456,A -85,B 0,C 180,E1 -12331.075,E2 -12331.075} C_VEL
LIN {X 0,Y 374.426,Z 402.113,A -85,B 0,C 180,E1 -12333.228,E2 -12333.228} C_VEL
LIN {X 0,Y 374.527,Z 399.407,A -85,B 0,C 180,E1 -12335.384,E2 -12335.384} C_VEL
LIN {X 0,Y 374.751,Z 395.259,A -85,B 0,C 180,E1 -12337.543,E2 -12337.543} C_VEL
LIN {X 0,Y 375.167,Z 389.548,A -85,B 0,C 180,E1 -12339.706,E2 -12339.706} C_VEL
LIN {X 0,Y 375.816,Z 383.113,A -85,B 0,C 180,E1 -12341.597,E2 -12341.597} C_VEL
LIN {X 0,Y 376.687,Z 375.12,A -85,B 0,C 180,E1 -12343.487,E2 -12343.487} C_VEL
LIN {X 0,Y 377.653,Z 366.761,A -85,B 0,C 180,E1 -12345.102,E2 -12345.102} C_VEL
LIN {X 0,Y 378.789,Z 356.699,A -85,B 0,C 180,E1 -12346.713,E2 -12346.713} C_VEL
LIN {X 0,Y 380.108,Z 345.476,A -85,B 0,C 180,E1 -12348.18,E2 -12348.18} C_VEL
LIN {X 0,Y 381.602,Z 332.887,A -85,B 0,C 180,E1 -12349.5,E2 -12349.5} C_VEL
LIN {X 0,Y 382.939,Z 319.599,A -85,B 0,C 180,E1 -12350.611,E2 -12350.611} C_VEL
LIN {X 0,Y 383.539,Z 310.88,A -85,B 0,C 180,E1 -12351.217,E2 -12351.217} C_VEL
LIN {X 0,Y 381.253,Z 296.827,A -85,B 0,C 180,E1 -12352.165,E2 -12352.165} C_VEL
LIN {X 0,Y 378.033,Z 282.461,A -85,B 0,C 180,E1 -12352.957,E2 -12352.957} C_VEL
LIN {X 0,Y 375.314,Z 272.317,A -85,B 0,C 180,E1 -12353.428,E2 -12353.428} C_VEL
LIN {X 0,Y 375.676,Z 266.987,A -85,B 0,C 180,E1 -12356.678,E2 -12356.678} C_VEL
LIN {X 0,Y 375.977,Z 263.109,A -85,B 0,C 180,E1 -12359.079,E2 -12359.079} C_VEL
LIN {X 0,Y 376.458,Z 257.198,A -85,B 0,C 180,E1 -12362.85,E2 -12362.85} C_VEL
LIN {X 0,Y 376.939,Z 251.312,A -85,B 0,C 180,E1 -12366.704,E2 -12366.704} C_VEL
LIN {X 0,Y 377.042,Z 247.519,A -85,B 0,C 180,E1 -12369.328,E2 -12369.328} C_VEL
LIN {X 0,Y 376.631,Z 243.629,A -85,B 0,C 180,E1 -12372.204,E2 -12372.204} C_VEL
LIN {X 0,Y 375.96,Z 239.284,A -85,B 0,C 180,E1 -12375.74,E2 -12375.74} C_VEL
LIN {X 0,Y 375.941,Z 239.284,A -85,B 0,C 180,E1 -12379.133,E2 -12379.133} C_VEL
LIN {X 0,Y 375.964,Z 239.281,A -85,B 0,C 180,E1 -12381.911,E2 -12381.911} C_VEL
LIN {X 0,Y 375.98,Z 239.279,A -85,B 0,C 180,E1 -12385.333,E2 -12385.333} C_VEL
LIN {X 0,Y 375.958,Z 239.28,A -85,B 0,C 180,E1 -12388.438,E2 -12388.438} C_VEL
LIN {X 0,Y 375.935,Z 239.284,A -85,B 0,C 180,E1 -12392.136,E2 -12392.136} C_VEL
LIN {X 0,Y 375.974,Z 239.28,A -85,B 0,C 180,E1 -12395.717,E2 -12395.717} C_VEL
LIN {X 0,Y 375.999,Z 239.275,A -85,B 0,C 180,E1 -12399.198,E2 -12399.198} C_VEL
LIN {X 0,Y 376.034,Z 239.269,A -85,B 0,C 180,E1 -12402.6,E2 -12402.6} C_VEL
LIN {X 0,Y 376.091,Z 239.26,A -85,B 0,C 180,E1 -12406.342,E2 -12406.342} C_VEL
LIN {X 0,Y 376.114,Z 239.259,A -85,B 0,C 180,E1 -12410.318,E2 -12410.318} C_VEL
LIN {X 0,Y 376.202,Z 239.251,A -85,B 0,C 180,E1 -12413.564,E2 -12413.564} C_VEL
LIN {X 0,Y 376.353,Z 239.229,A -85,B 0,C 180,E1 -12417.86,E2 -12417.86} C_VEL
LIN {X 0,Y 376.483,Z 239.216,A -85,B 0,C 180,E1 -12420,E2 -12420} C_VEL
LIN {X 0,Y 376.35,Z 239.23,A -85,B 0,C 180,E1 -12422.14,E2 -12422.14} C_VEL
LIN {X 0,Y 376.223,Z 239.246,A -85,B 0,C 180,E1 -12426.649,E2 -12426.649} C_VEL
LIN {X 0,Y 376.121,Z 239.26,A -85,B 0,C 180,E1 -12429.682,E2 -12429.682} C_VEL
LIN {X 0,Y 376.091,Z 239.26,A -85,B 0,C 180,E1 -12433.658,E2 -12433.658} C_VEL
LIN {X 0,Y 376.046,Z 239.27,A -85,B 0,C 180,E1 -12437.608,E2 -12437.608} C_VEL
LIN {X 0,Y 375.98,Z 239.277,A -85,B 0,C 180,E1 -12440.832,E2 -12440.832} C_VEL
LIN {X 0,Y 375.99,Z 239.276,A -85,B 0,C 180,E1 -12444.282,E2 -12444.282} C_VEL
LIN {X 0,Y 376.021,Z 239.27,A -85,B 0,C 180,E1 -12446.652,E2 -12446.652} C_VEL
LIN {X 0,Y 375.966,Z 239.278,A -85,B 0,C 180,E1 -12450.313,E2 -12450.313} C_VEL
LIN {X 0,Y 375.961,Z 239.281,A -85,B 0,C 180,E1 -12454.111,E2 -12454.111} C_VEL
LIN {X 0,Y 375.954,Z 239.28,A -85,B 0,C 180,E1 -12456.741,E2 -12456.741} C_VEL
LIN {X 0,Y 375.94,Z 239.28,A -85,B 0,C 180,E1 -12459.962,E2 -12459.962} C_VEL
LIN {X 0,Y 375.93,Z 239.286,A -85,B 0,C 180,E1 -12463.766,E2 -12463.766} C_VEL
LIN {X 0,Y 375.935,Z 239.285,A -85,B 0,C 180,E1 -12466.811,E2 -12466.811} C_VEL
LIN {X 0,Y 375.948,Z 239.538,A -85,B 0,C 180,E1 -12469.134,E2 -12469.134} C_VEL
LIN {X 0,Y 376.121,Z 242.516,A -85,B 0,C 180,E1 -12471.93,E2 -12471.93} C_VEL
LIN {X 0,Y 376.011,Z 245.447,A -85,B 0,C 180,E1 -12474.59,E2 -12474.59} C_VEL
LIN {X 0,Y 375.719,Z 249.872,A -85,B 0,C 180,E1 -12478.416,E2 -12478.416} C_VEL
LIN {X 0,Y 375.43,Z 254.367,A -85,B 0,C 180,E1 -12482.096,E2 -12482.096} C_VEL
LIN {X 0,Y 375.222,Z 258.849,A -85,B 0,C 180,E1 -12485.665,E2 -12485.665} C_VEL
LIN {X 0,Y 375.178,Z 260.078,A -85,B 0,C 180,E1 -12486.62,E2 -12486.62} C_VEL
LIN {X 0,Y 379.984,Z 276.386,A -85,B 0,C 180,E1 -12487.48,E2 -12487.48} C_VEL
LIN {X 0,Y 383.009,Z 289.191,A -85,B 0,C 180,E1 -12488.297,E2 -12488.297} C_VEL
LIN {X 0,Y 384.162,Z 295.325,A -85,B 0,C 180,E1 -12488.738,E2 -12488.738} C_VEL
LIN {X 0,Y 383.205,Z 307.968,A -85,B 0,C 180,E1 -12489.607,E2 -12489.607} C_VEL
LIN {X 0,Y 382.001,Z 320.188,A -85,B 0,C 180,E1 -12490.661,E2 -12490.661} C_VEL
LIN {X 0,Y 380.619,Z 332.506,A -85,B 0,C 180,E1 -12491.984,E2 -12491.984} C_VEL
LIN {X 0,Y 379.41,Z 342.628,A -85,B 0,C 180,E1 -12493.315,E2 -12493.315} C_VEL
LIN {X 0,Y 378.124,Z 352.672,A -85,B 0,C 180,E1 -12494.917,E2 -12494.917} C_VEL
LIN {X 0,Y 377.218,Z 361.007,A -85,B 0,C 180,E1 -12496.533,E2 -12496.533} C_VEL
LIN {X 0,Y 376.169,Z 368.969,A -85,B 0,C 180,E1 -12498.414,E2 -12498.414} C_VEL
LIN {X 0,Y 375.514,Z 375.373,A -85,B 0,C 180,E1 -12500.303,E2 -12500.303} C_VEL
LIN {X 0,Y 374.994,Z 381.051,A -85,B 0,C 180,E1 -12502.462,E2 -12502.462} C_VEL
LIN {X 0,Y 374.734,Z 385.177,A -85,B 0,C 180,E1 -12504.619,E2 -12504.619} C_VEL
LIN {X 0,Y 374.502,Z 387.877,A -85,B 0,C 180,E1 -12506.773,E2 -12506.773} C_VEL
LIN {X 0,Y 374.476,Z 389.228,A -85,B 0,C 180,E1 -12508.925,E2 -12508.925} C_VEL
LIN {X 0,Y 374.476,Z 389.263,A -85,B 0,C 180,E1 -12511.075,E2 -12511.075} C_VEL
LIN {X 0,Y 374.501,Z 387.976,A -85,B 0,C 180,E1 -12513.228,E2 -12513.228} C_VEL
LIN {X 0,Y 374.726,Z 385.335,A -85,B 0,C 180,E1 -12515.381,E2 -12515.381} C_VEL
LIN {X 0,Y 374.991,Z 381.277,A -85,B 0,C 180,E1 -12517.539,E2 -12517.539} C_VEL
LIN {X 0,Y 375.493,Z 375.668,A -85,B 0,C 180,E1 -12519.698,E2 -12519.698} C_VEL
LIN {X 0,Y 376.129,Z 369.334,A -85,B 0,C 180,E1 -12521.588,E2 -12521.588} C_VEL
LIN {X 0,Y 377.201,Z 361.452,A -85,B 0,C 180,E1 -12523.468,E2 -12523.468} C_VEL
LIN {X 0,Y 378.067,Z 353.21,A -85,B 0,C 180,E1 -12525.085,E2 -12525.085} C_VEL
LIN {X 0,Y 379.363,Z 343.271,A -85,B 0,C 180,E1 -12526.688,E2 -12526.688} C_VEL
LIN {X 0,Y 380.667,Z 332.207,A -85,B 0,C 180,E1 -12528.153,E2 -12528.153} C_VEL
LIN {X 0,Y 381.926,Z 321.187,A -85,B 0,C 180,E1 -12529.343,E2 -12529.343} C_VEL
LIN {X 0,Y 383.119,Z 309.223,A -85,B 0,C 180,E1 -12530.398,E2 -12530.398} C_VEL
LIN {X 0,Y 384.211,Z 295.723,A -85,B 0,C 180,E1 -12531.336,E2 -12531.336} C_VEL
LIN {X 0,Y 381.554,Z 282.584,A -85,B 0,C 180,E1 -12532.243,E2 -12532.243} C_VEL
LIN {X 0,Y 379.768,Z 275.602,A -85,B 0,C 180,E1 -12532.667,E2 -12532.667} C_VEL
LIN {X 0,Y 378.291,Z 273.784,A -85,B 0,C 180,E1 -12532.835,E2 -12532.835} C_VEL
LIN {X 0,Y 372.162,Z 271.072,A -85,B 0,C 180,E1 -12533.343,E2 -12533.343} C_VEL
LIN {X 0,Y 370.96,Z 269.427,A -85,B 0,C 180,E1 -12533.478,E2 -12533.478} C_VEL
LIN {X 0,Y 368.158,Z 260.199,A -85,B 0,C 180,E1 -12533.963,E2 -12533.963} C_VEL
LIN {X 0,Y 368.324,Z 256.121,A -85,B 0,C 180,E1 -12537.255,E2 -12537.255} C_VEL
LIN {X 0,Y 368.637,Z 251.622,A -85,B 0,C 180,E1 -12540.981,E2 -12540.981} C_VEL
LIN {X 0,Y 368.974,Z 247.149,A -85,B 0,C 180,E1 -12544.85,E2 -12544.85} C_VEL
LIN {X 0,Y 369.071,Z 244.208,A -85,B 0,C 180,E1 -12547.543,E2 -12547.543} C_VEL
LIN {X 0,Y 368.984,Z 241.23,A -85,B 0,C 180,E1 -12550.37,E2 -12550.37} C_VEL
LIN {X 0,Y 368.873,Z 240.163,A -85,B 0,C 180,E1 -12552.008,E2 -12552.008} C_VEL
LIN {X 0,Y 368.881,Z 240.163,A -85,B 0,C 180,E1 -12555.176,E2 -12555.176} C_VEL
LIN {X 0,Y 368.871,Z 240.165,A -85,B 0,C 180,E1 -12558.176,E2 -12558.176} C_VEL
LIN {X 0,Y 368.88,Z 240.163,A -85,B 0,C 180,E1 -12561.366,E2 -12561.366} C_VEL
LIN {X 0,Y 368.939,Z 240.153,A -85,B 0,C 180,E1 -12565.147,E2 -12565.147} C_VEL
LIN {X 0,Y 368.932,Z 240.156,A -85,B 0,C 180,E1 -12569.047,E2 -12569.047} C_VEL
LIN {X 0,Y 368.966,Z 240.152,A -85,B 0,C 180,E1 -12572.797,E2 -12572.797} C_VEL
LIN {X 0,Y 368.937,Z 240.154,A -85,B 0,C 180,E1 -12576.117,E2 -12576.117} C_VEL
LIN {X 0,Y 368.939,Z 240.151,A -85,B 0,C 180,E1 -12579.947,E2 -12579.947} C_VEL
LIN {X 0,Y 368.979,Z 240.149,A -85,B 0,C 180,E1 -12583.399,E2 -12583.399} C_VEL
LIN {X 0,Y 369.061,Z 240.139,A -85,B 0,C 180,E1 -12586.79,E2 -12586.79} C_VEL
LIN {X 0,Y 369.066,Z 240.138,A -85,B 0,C 180,E1 -12590.132,E2 -12590.132} C_VEL
LIN {X 0,Y 369.191,Z 240.124,A -85,B 0,C 180,E1 -12593.441,E2 -12593.441} C_VEL
LIN {X 0,Y 369.316,Z 240.105,A -85,B 0,C 180,E1 -12597.819,E2 -12597.819} C_VEL
LIN {X 0,Y 369.248,Z 240.114,A -85,B 0,C 180,E1 -12601.091,E2 -12601.091} C_VEL
LIN {X 0,Y 369.319,Z 240.104,A -85,B 0,C 180,E1 -12602.181,E2 -12602.181} C_VEL
LIN {X 0,Y 369.163,Z 240.128,A -85,B 0,C 180,E1 -12606.559,E2 -12606.559} C_VEL
LIN {X 0,Y 369.065,Z 240.139,A -85,B 0,C 180,E1 -12609.868,E2 -12609.868} C_VEL
LIN {X 0,Y 369.04,Z 240.141,A -85,B 0,C 180,E1 -12613.772,E2 -12613.772} C_VEL
LIN {X 0,Y 368.993,Z 240.149,A -85,B 0,C 180,E1 -12617.743,E2 -12617.743} C_VEL
LIN {X 0,Y 368.912,Z 240.159,A -85,B 0,C 180,E1 -12621.221,E2 -12621.221} C_VEL
LIN {X 0,Y 368.928,Z 240.152,A -85,B 0,C 180,E1 -12624.777,E2 -12624.777} C_VEL
LIN {X 0,Y 368.897,Z 240.159,A -85,B 0,C 180,E1 -12628.793,E2 -12628.793} C_VEL
LIN {X 0,Y 368.9,Z 240.159,A -85,B 0,C 180,E1 -12632.238,E2 -12632.238} C_VEL
LIN {X 0,Y 368.931,Z 240.157,A -85,B 0,C 180,E1 -12635.001,E2 -12635.001} C_VEL
LIN {X 0,Y 368.909,Z 240.16,A -85,B 0,C 180,E1 -12638.64,E2 -12638.64} C_VEL
LIN {X 0,Y 368.883,Z 240.165,A -85,B 0,C 180,E1 -12642.009,E2 -12642.009} C_VEL
LIN {X 0,Y 368.942,Z 240.365,A -85,B 0,C 180,E1 -12644.163,E2 -12644.163} C_VEL
LIN {X 0,Y 369.682,Z 244.939,A -85,B 0,C 180,E1 -12647.853,E2 -12647.853} C_VEL
LIN {X 0,Y 369.978,Z 247.471,A -85,B 0,C 180,E1 -12649.77,E2 -12649.77} C_VEL
LIN {X 0,Y 369.976,Z 251.373,A -85,B 0,C 180,E1 -12652.564,E2 -12652.564} C_VEL
LIN {X 0,Y 369.644,Z 255.268,A -85,B 0,C 180,E1 -12655.223,E2 -12655.223} C_VEL
LIN {X 0,Y 369.307,Z 259.16,A -85,B 0,C 180,E1 -12657.802,E2 -12657.802} C_VEL
LIN {X 0,Y 368.899,Z 264.944,A -85,B 0,C 180,E1 -12661.557,E2 -12661.557} C_VEL
LIN {X 0,Y 368.363,Z 270.735,A -85,B 0,C 180,E1 -12665.182,E2 -12665.182} C_VEL
LIN {X 0,Y 368.294,Z 272.22,A -85,B 0,C 180,E1 -12666.099,E2 -12666.099} C_VEL
LIN {X 0,Y 372.088,Z 286.413,A -85,B 0,C 180,E1 -12666.79,E2 -12666.79} C_VEL
LIN {X 0,Y 374.895,Z 299.636,A -85,B 0,C 180,E1 -12667.583,E2 -12667.583} C_VEL
LIN {X 0,Y 376.873,Z 312.907,A -85,B 0,C 180,E1 -12668.533,E2 -12668.533} C_VEL
LIN {X 0,Y 375.638,Z 326.165,A -85,B 0,C 180,E1 -12669.533,E2 -12669.533} C_VEL
LIN {X 0,Y 374.272,Z 338.194,A -85,B 0,C 180,E1 -12670.673,E2 -12670.673} C_VEL
LIN {X 0,Y 372.864,Z 349.74,A -85,B 0,C 180,E1 -12672.022,E2 -12672.022} C_VEL
LIN {X 0,Y 371.535,Z 360.203,A -85,B 0,C 180,E1 -12673.516,E2 -12673.516} C_VEL
LIN {X 0,Y 370.354,Z 369.95,A -85,B 0,C 180,E1 -12675.212,E2 -12675.212} C_VEL
LIN {X 0,Y 369.354,Z 378.672,A -85,B 0,C 180,E1 -12677.081,E2 -12677.081} C_VEL
LIN {X 0,Y 368.434,Z 385.951,A -85,B 0,C 180,E1 -12679.003,E2 -12679.003} C_VEL
LIN {X 0,Y 367.977,Z 391.058,A -85,B 0,C 180,E1 -12680.657,E2 -12680.657} C_VEL
LIN {X 0,Y 367.649,Z 396.33,A -85,B 0,C 180,E1 -12682.862,E2 -12682.862} C_VEL
LIN {X 0,Y 367.451,Z 399.282,A -85,B 0,C 180,E1 -12684.512,E2 -12684.512} C_VEL
LIN {X 0,Y 367.345,Z 401.985,A -85,B 0,C 180,E1 -12686.71,E2 -12686.71} C_VEL
LIN {X 0,Y 367.352,Z 403.324,A -85,B 0,C 180,E1 -12688.904,E2 -12688.904} C_VEL
LIN {X 0,Y 367.352,Z 403.321,A -85,B 0,C 180,E1 -12691.096,E2 -12691.096} C_VEL
LIN {X 0,Y 367.345,Z 401.978,A -85,B 0,C 180,E1 -12693.29,E2 -12693.29} C_VEL
LIN {X 0,Y 367.445,Z 399.271,A -85,B 0,C 180,E1 -12695.488,E2 -12695.488} C_VEL
LIN {X 0,Y 367.679,Z 395.123,A -85,B 0,C 180,E1 -12697.689,E2 -12697.689} C_VEL
LIN {X 0,Y 368.132,Z 389.411,A -85,B 0,C 180,E1 -12699.894,E2 -12699.894} C_VEL
LIN {X 0,Y 368.831,Z 382.976,A -85,B 0,C 180,E1 -12701.82,E2 -12701.82} C_VEL
LIN {X 0,Y 369.757,Z 374.983,A -85,B 0,C 180,E1 -12703.744,E2 -12703.744} C_VEL
LIN {X 0,Y 370.739,Z 366.623,A -85,B 0,C 180,E1 -12705.39,E2 -12705.39} C_VEL
LIN {X 0,Y 371.95,Z 356.561,A -85,B 0,C 180,E1 -12707.03,E2 -12707.03} C_VEL
LIN {X 0,Y 373.35,Z 345.337,A -85,B 0,C 180,E1 -12708.521,E2 -12708.521} C_VEL
LIN {X 0,Y 374.871,Z 332.841,A -85,B 0,C 180,E1 -12709.856,E2 -12709.856} C_VEL
LIN {X 0,Y 376.197,Z 320.427,A -85,B 0,C 180,E1 -12710.919,E2 -12710.919} C_VEL
LIN {X 0,Y 376.746,Z 311.736,A -85,B 0,C 180,E1 -12711.546,E2 -12711.546} C_VEL
LIN {X 0,Y 374.849,Z 299.598,A -85,B 0,C 180,E1 -12712.409,E2 -12712.409} C_VEL
LIN {X 0,Y 371.799,Z 285.181,A -85,B 0,C 180,E1 -12713.265,E2 -12713.265} C_VEL
LIN {X 0,Y 368.282,Z 272.213,A -85,B 0,C 180,E1 -12713.892,E2 -12713.892} C_VEL
LIN {X 0,Y 368.684,Z 266.841,A -85,B 0,C 180,E1 -12717.226,E2 -12717.226} C_VEL
LIN {X 0,Y 369.007,Z 262.993,A -85,B 0,C 180,E1 -12719.682,E2 -12719.682} C_VEL
LIN {X 0,Y 369.472,Z 257.192,A -85,B 0,C 180,E1 -12723.479,E2 -12723.479} C_VEL
LIN {X 0,Y 369.946,Z 251.85,A -85,B 0,C 180,E1 -12727.071,E2 -12727.071} C_VEL
LIN {X 0,Y 370.05,Z 249.303,A -85,B 0,C 180,E1 -12728.861,E2 -12728.861} C_VEL
LIN {X 0,Y 369.721,Z 245.48,A -85,B 0,C 180,E1 -12731.706,E2 -12731.706} C_VEL
LIN {X 0,Y 369.067,Z 241.079,A -85,B 0,C 180,E1 -12735.205,E2 -12735.205} C_VEL
LIN {X 0,Y 368.895,Z 240.165,A -85,B 0,C 180,E1 -12736.152,E2 -12736.152} C_VEL
LIN {X 0,Y 368.912,Z 240.16,A -85,B 0,C 180,E1 -12739.643,E2 -12739.643} C_VEL
LIN {X 0,Y 368.902,Z 240.162,A -85,B 0,C 180,E1 -12743.144,E2 -12743.144} C_VEL
LIN {X 0,Y 368.897,Z 240.161,A -85,B 0,C 180,E1 -12746.462,E2 -12746.462} C_VEL
LIN {X 0,Y 368.93,Z 240.158,A -85,B 0,C 180,E1 -12749.047,E2 -12749.047} C_VEL
LIN {X 0,Y 368.872,Z 240.162,A -85,B 0,C 180,E1 -12752.789,E2 -12752.789} C_VEL
LIN {X 0,Y 368.95,Z 240.152,A -85,B 0,C 180,E1 -12756.421,E2 -12756.421} C_VEL
LIN {X 0,Y 368.937,Z 240.154,A -85,B 0,C 180,E1 -12759.947,E2 -12759.947} C_VEL
LIN {X 0,Y 368.97,Z 240.149,A -85,B 0,C 180,E1 -12763.399,E2 -12763.399} C_VEL
LIN {X 0,Y 369.059,Z 240.138,A -85,B 0,C 180,E1 -12766.79,E2 -12766.79} C_VEL
LIN {X 0,Y 369.064,Z 240.135,A -85,B 0,C 180,E1 -12770.132,E2 -12770.132} C_VEL
LIN {X 0,Y 369.162,Z 240.128,A -85,B 0,C 180,E1 -12773.441,E2 -12773.441} C_VEL
LIN {X 0,Y 369.318,Z 240.105,A -85,B 0,C 180,E1 -12777.819,E2 -12777.819} C_VEL
LIN {X 0,Y 369.432,Z 240.094,A -85,B 0,C 180,E1 -12780,E2 -12780} C_VEL
LIN {X 0,Y 369.315,Z 240.106,A -85,B 0,C 180,E1 -12782.181,E2 -12782.181} C_VEL
LIN {X 0,Y 369.193,Z 240.122,A -85,B 0,C 180,E1 -12786.635,E2 -12786.635} C_VEL
LIN {X 0,Y 369.069,Z 240.14,A -85,B 0,C 180,E1 -12789.868,E2 -12789.868} C_VEL
LIN {X 0,Y 369.039,Z 240.139,A -85,B 0,C 180,E1 -12793.772,E2 -12793.772} C_VEL
LIN {X 0,Y 369.003,Z 240.147,A -85,B 0,C 180,E1 -12797.768,E2 -12797.768} C_VEL
LIN {X 0,Y 368.911,Z 240.158,A -85,B 0,C 180,E1 -12801.221,E2 -12801.221} C_VEL
LIN {X 0,Y 368.956,Z 240.151,A -85,B 0,C 180,E1 -12804.776,E2 -12804.776} C_VEL
LIN {X 0,Y 368.965,Z 240.15,A -85,B 0,C 180,E1 -12807.203,E2 -12807.203} C_VEL
LIN {X 0,Y 368.931,Z 240.156,A -85,B 0,C 180,E1 -12810.954,E2 -12810.954} C_VEL
LIN {X 0,Y 368.93,Z 240.154,A -85,B 0,C 180,E1 -12815.001,E2 -12815.001} C_VEL
LIN {X 0,Y 368.879,Z 240.162,A -85,B 0,C 180,E1 -12818.634,E2 -12818.634} C_VEL
LIN {X 0,Y 368.871,Z 240.164,A -85,B 0,C 180,E1 -12822.008,E2 -12822.008} C_VEL
LIN {X 0,Y 368.88,Z 240.163,A -85,B 0,C 180,E1 -12825.176,E2 -12825.176} C_VEL
LIN {X 0,Y 368.876,Z 240.165,A -85,B 0,C 180,E1 -12828.177,E2 -12828.177} C_VEL
LIN {X 0,Y 368.985,Z 241.113,A -85,B 0,C 180,E1 -12829.64,E2 -12829.64} C_VEL
LIN {X 0,Y 369.081,Z 244.094,A -85,B 0,C 180,E1 -12832.458,E2 -12832.458} C_VEL
LIN {X 0,Y 368.968,Z 247.035,A -85,B 0,C 180,E1 -12835.15,E2 -12835.15} C_VEL
LIN {X 0,Y 368.63,Z 251.574,A -85,B 0,C 180,E1 -12839.086,E2 -12839.086} C_VEL
LIN {X 0,Y 368.316,Z 255.991,A -85,B 0,C 180,E1 -12842.745,E2 -12842.745} C_VEL
LIN {X 0,Y 368.128,Z 260.217,A -85,B 0,C 180,E1 -12846.154,E2 -12846.154} C_VEL
LIN {X 0,Y 372.816,Z 275.839,A -85,B 0,C 180,E1 -12846.994,E2 -12846.994} C_VEL
LIN {X 0,Y 375.968,Z 288.7,A -85,B 0,C 180,E1 -12847.833,E2 -12847.833} C_VEL
LIN {X 0,Y 377.472,Z 297.428,A -85,B 0,C 180,E1 -12848.471,E2 -12848.471} C_VEL
LIN {X 0,Y 376.397,Z 309.824,A -85,B 0,C 180,E1 -12849.364,E2 -12849.364} C_VEL
LIN {X 0,Y 375.16,Z 321.693,A -85,B 0,C 180,E1 -12850.436,E2 -12850.436} C_VEL
LIN {X 0,Y 373.739,Z 333.711,A -85,B 0,C 180,E1 -12851.782,E2 -12851.782} C_VEL
LIN {X 0,Y 372.348,Z 344.543,A -85,B 0,C 180,E1 -12853.271,E2 -12853.271} C_VEL
LIN {X 0,Y 371.042,Z 354.216,A -85,B 0,C 180,E1 -12854.89,E2 -12854.89} C_VEL
LIN {X 0,Y 370.138,Z 362.37,A -85,B 0,C 180,E1 -12856.55,E2 -12856.55} C_VEL
LIN {X 0,Y 369.095,Z 370.107,A -85,B 0,C 180,E1 -12858.467,E2 -12858.467} C_VEL
LIN {X 0,Y 368.5,Z 375.51,A -85,B 0,C 180,E1 -12860.116,E2 -12860.116} C_VEL
LIN {X 0,Y 367.928,Z 381.188,A -85,B 0,C 180,E1 -12862.316,E2 -12862.316} C_VEL
LIN {X 0,Y 367.646,Z 385.313,A -85,B 0,C 180,E1 -12864.515,E2 -12864.515} C_VEL
LIN {X 0,Y 367.419,Z 388.012,A -85,B 0,C 180,E1 -12866.71,E2 -12866.71} C_VEL
LIN {X 0,Y 367.377,Z 389.363,A -85,B 0,C 180,E1 -12868.904,E2 -12868.904} C_VEL
LIN {X 0,Y 367.377,Z 389.397,A -85,B 0,C 180,E1 -12871.096,E2 -12871.096} C_VEL
LIN {X 0,Y 367.418,Z 388.11,A -85,B 0,C 180,E1 -12873.29,E2 -12873.29} C_VEL
LIN {X 0,Y 367.64,Z 385.469,A -85,B 0,C 180,E1 -12875.485,E2 -12875.485} C_VEL
LIN {X 0,Y 367.865,Z 382.567,A -85,B 0,C 180,E1 -12877.134,E2 -12877.134} C_VEL
LIN {X 0,Y 368.32,Z 377.392,A -85,B 0,C 180,E1 -12879.334,E2 -12879.334} C_VEL
LIN {X 0,Y 368.869,Z 372.363,A -85,B 0,C 180,E1 -12880.984,E2 -12880.984} C_VEL
LIN {X 0,Y 369.793,Z 365.179,A -85,B 0,C 180,E1 -12882.904,E2 -12882.904} C_VEL
LIN {X 0,Y 370.582,Z 357.722,A -85,B 0,C 180,E1 -12884.54,E2 -12884.54} C_VEL
LIN {X 0,Y 371.805,Z 348.61,A -85,B 0,C 180,E1 -12886.189,E2 -12886.189} C_VEL
LIN {X 0,Y 373.257,Z 337.652,A -85,B 0,C 180,E1 -12887.817,E2 -12887.817} C_VEL
LIN {X 0,Y 374.654,Z 326.474,A -85,B 0,C 180,E1 -12889.164,E2 -12889.164} C_VEL
LIN {X 0,Y 375.999,Z 314.103,A -85,B 0,C 180,E1 -12890.373,E2 -12890.373} C_VEL
LIN {X 0,Y 377.125,Z 301.663,A -85,B 0,C 180,E1 -12891.347,E2 -12891.347} C_VEL
LIN {X 0,Y 377.435,Z 295.974,A -85,B 0,C 180,E1 -12891.73,E2 -12891.73} C_VEL
LIN {X 0,Y 374.397,Z 281.791,A -85,B 0,C 180,E1 -12892.736,E2 -12892.736} C_VEL
LIN {X 0,Y 370.96,Z 269.427,A -85,B 0,C 180,E1 -12893.478,E2 -12893.478} C_VEL
LIN {X 0,Y 369.286,Z 266.064,A -85,B 0,C 180,E1 -12893.739,E2 -12893.739} C_VEL
LIN {X 0,Y 366.142,Z 262.754,A -85,B 0,C 180,E1 -12894.24,E2 -12894.24} C_VEL
LIN {X 0,Y 363.092,Z 260.455,A -85,B 0,C 180,E1 -12894.885,E2 -12894.885} C_VEL
LIN {X 0,Y 361.53,Z 259.214,A -85,B 0,C 180,E1 -12895.462,E2 -12895.462} C_VEL
LIN {X 0,Y 361.178,Z 258.598,A -85,B 0,C 180,E1 -12895.883,E2 -12895.883} C_VEL
LIN {X 0,Y 361.413,Z 254.755,A -85,B 0,C 180,E1 -12899.088,E2 -12899.088} C_VEL
LIN {X 0,Y 361.614,Z 251.738,A -85,B 0,C 180,E1 -12901.652,E2 -12901.652} C_VEL
LIN {X 0,Y 361.952,Z 247.557,A -85,B 0,C 180,E1 -12905.362,E2 -12905.362} C_VEL
LIN {X 0,Y 362.048,Z 244.304,A -85,B 0,C 180,E1 -12908.403,E2 -12908.403} C_VEL
LIN {X 0,Y 361.831,Z 241.336,A -85,B 0,C 180,E1 -12911.331,E2 -12911.331} C_VEL
LIN {X 0,Y 361.836,Z 241.041,A -85,B 0,C 180,E1 -12912.829,E2 -12912.829} C_VEL
LIN {X 0,Y 361.82,Z 241.044,A -85,B 0,C 180,E1 -12915.947,E2 -12915.947} C_VEL
LIN {X 0,Y 361.814,Z 241.043,A -85,B 0,C 180,E1 -12919.249,E2 -12919.249} C_VEL
LIN {X 0,Y 361.867,Z 241.037,A -85,B 0,C 180,E1 -12922.982,E2 -12922.982} C_VEL
LIN {X 0,Y 361.861,Z 241.035,A -85,B 0,C 180,E1 -12926.631,E2 -12926.631} C_VEL
LIN {X 0,Y 361.875,Z 241.034,A -85,B 0,C 180,E1 -12929.672,E2 -12929.672} C_VEL
LIN {X 0,Y 361.957,Z 241.023,A -85,B 0,C 180,E1 -12933.475,E2 -12933.475} C_VEL
LIN {X 0,Y 361.882,Z 241.034,A -85,B 0,C 180,E1 -12937.144,E2 -12937.144} C_VEL
LIN {X 0,Y 361.909,Z 241.031,A -85,B 0,C 180,E1 -12940.723,E2 -12940.723} C_VEL
LIN {X 0,Y 361.936,Z 241.025,A -85,B 0,C 180,E1 -12943.066,E2 -12943.066} C_VEL
LIN {X 0,Y 362.002,Z 241.017,A -85,B 0,C 180,E1 -12946.528,E2 -12946.528} C_VEL
LIN {X 0,Y 362.003,Z 241.016,A -85,B 0,C 180,E1 -12949.937,E2 -12949.937} C_VEL
LIN {X 0,Y 362.152,Z 241,A -85,B 0,C 180,E1 -12953.313,E2 -12953.313} C_VEL
LIN {X 0,Y 362.28,Z 240.981,A -85,B 0,C 180,E1 -12957.776,E2 -12957.776} C_VEL
LIN {X 0,Y 362.216,Z 240.991,A -85,B 0,C 180,E1 -12961.112,E2 -12961.112} C_VEL
LIN {X 0,Y 362.283,Z 240.98,A -85,B 0,C 180,E1 -12962.223,E2 -12962.223} C_VEL
LIN {X 0,Y 362.126,Z 241.003,A -85,B 0,C 180,E1 -12966.687,E2 -12966.687} C_VEL
LIN {X 0,Y 362.002,Z 241.019,A -85,B 0,C 180,E1 -12970.063,E2 -12970.063} C_VEL
LIN {X 0,Y 362.001,Z 241.018,A -85,B 0,C 180,E1 -12973.899,E2 -12973.899} C_VEL
LIN {X 0,Y 361.931,Z 241.026,A -85,B 0,C 180,E1 -12976.934,E2 -12976.934} C_VEL
LIN {X 0,Y 361.889,Z 241.031,A -85,B 0,C 180,E1 -12980.461,E2 -12980.461} C_VEL
LIN {X 0,Y 361.895,Z 241.032,A -85,B 0,C 180,E1 -12984.113,E2 -12984.113} C_VEL
LIN {X 0,Y 361.842,Z 241.038,A -85,B 0,C 180,E1 -12987.785,E2 -12987.785} C_VEL
LIN {X 0,Y 361.848,Z 241.035,A -85,B 0,C 180,E1 -12991.285,E2 -12991.285} C_VEL
LIN {X 0,Y 361.856,Z 241.04,A -85,B 0,C 180,E1 -12994.28,E2 -12994.28} C_VEL
LIN {X 0,Y 361.865,Z 241.039,A -85,B 0,C 180,E1 -12997.223,E2 -12997.223} C_VEL
LIN {X 0,Y 361.837,Z 241.041,A -85,B 0,C 180,E1 -13000.755,E2 -13000.755} C_VEL
LIN {X 0,Y 361.867,Z 241.193,A -85,B 0,C 180,E1 -13003.771,E2 -13003.771} C_VEL
LIN {X 0,Y 362.6,Z 245.626,A -85,B 0,C 180,E1 -13007.436,E2 -13007.436} C_VEL
LIN {X 0,Y 362.977,Z 249.315,A -85,B 0,C 180,E1 -13010.286,E2 -13010.286} C_VEL
LIN {X 0,Y 362.882,Z 253.206,A -85,B 0,C 180,E1 -13013.102,E2 -13013.102} C_VEL
LIN {X 0,Y 362.358,Z 259.044,A -85,B 0,C 180,E1 -13017.107,E2 -13017.107} C_VEL
LIN {X 0,Y 361.902,Z 264.807,A -85,B 0,C 180,E1 -13020.955,E2 -13020.955} C_VEL
LIN {X 0,Y 361.365,Z 270.59,A -85,B 0,C 180,E1 -13024.668,E2 -13024.668} C_VEL
LIN {X 0,Y 361.26,Z 272.115,A -85,B 0,C 180,E1 -13025.605,E2 -13025.605} C_VEL
LIN {X 0,Y 365.24,Z 286.803,A -85,B 0,C 180,E1 -13026.35,E2 -13026.35} C_VEL
LIN {X 0,Y 368.041,Z 299.974,A -85,B 0,C 180,E1 -13027.169,E2 -13027.169} C_VEL
LIN {X 0,Y 369.921,Z 311.774,A -85,B 0,C 180,E1 -13028.035,E2 -13028.035} C_VEL
LIN {X 0,Y 369.911,Z 316.906,A -85,B 0,C 180,E1 -13028.416,E2 -13028.416} C_VEL
LIN {X 0,Y 368.616,Z 329.385,A -85,B 0,C 180,E1 -13029.442,E2 -13029.442} C_VEL
LIN {X 0,Y 367.052,Z 341.772,A -85,B 0,C 180,E1 -13030.714,E2 -13030.714} C_VEL
LIN {X 0,Y 365.674,Z 352.645,A -85,B 0,C 180,E1 -13032.091,E2 -13032.091} C_VEL
LIN {X 0,Y 364.247,Z 363.392,A -85,B 0,C 180,E1 -13033.753,E2 -13033.753} C_VEL
LIN {X 0,Y 363.122,Z 372.269,A -85,B 0,C 180,E1 -13035.427,E2 -13035.427} C_VEL
LIN {X 0,Y 362.115,Z 380.779,A -85,B 0,C 180,E1 -13037.388,E2 -13037.388} C_VEL
LIN {X 0,Y 361.251,Z 387.636,A -85,B 0,C 180,E1 -13039.349,E2 -13039.349} C_VEL
LIN {X 0,Y 360.816,Z 392.364,A -85,B 0,C 180,E1 -13041.035,E2 -13041.035} C_VEL
LIN {X 0,Y 360.496,Z 397.265,A -85,B 0,C 180,E1 -13043.282,E2 -13043.282} C_VEL
LIN {X 0,Y 360.328,Z 400.673,A -85,B 0,C 180,E1 -13045.525,E2 -13045.525} C_VEL
LIN {X 0,Y 360.231,Z 402.688,A -85,B 0,C 180,E1 -13047.764,E2 -13047.764} C_VEL
LIN {X 0,Y 360.29,Z 403.355,A -85,B 0,C 180,E1 -13050,E2 -13050} C_VEL
LIN {X 0,Y 360.231,Z 402.683,A -85,B 0,C 180,E1 -13052.236,E2 -13052.236} C_VEL
LIN {X 0,Y 360.325,Z 400.664,A -85,B 0,C 180,E1 -13054.475,E2 -13054.475} C_VEL
LIN {X 0,Y 360.495,Z 397.248,A -85,B 0,C 180,E1 -13056.717,E2 -13056.717} C_VEL
LIN {X 0,Y 360.815,Z 392.335,A -85,B 0,C 180,E1 -13058.965,E2 -13058.965} C_VEL
LIN {X 0,Y 361.25,Z 387.599,A -85,B 0,C 180,E1 -13060.651,E2 -13060.651} C_VEL
LIN {X 0,Y 362.106,Z 380.735,A -85,B 0,C 180,E1 -13062.612,E2 -13062.612} C_VEL
LIN {X 0,Y 363.122,Z 372.214,A -85,B 0,C 180,E1 -13064.573,E2 -13064.573} C_VEL
LIN {X 0,Y 364.237,Z 363.325,A -85,B 0,C 180,E1 -13066.247,E2 -13066.247} C_VEL
LIN {X 0,Y 365.665,Z 352.562,A -85,B 0,C 180,E1 -13067.91,E2 -13067.91} C_VEL
LIN {X 0,Y 367.041,Z 341.671,A -85,B 0,C 180,E1 -13069.287,E2 -13069.287} C_VEL
LIN {X 0,Y 368.669,Z 329.11,A -85,B 0,C 180,E1 -13070.571,E2 -13070.571} C_VEL
LIN {X 0,Y 369.912,Z 316.563,A -85,B 0,C 180,E1 -13071.598,E2 -13071.598} C_VEL
LIN {X 0,Y 369.993,Z 312.591,A -85,B 0,C 180,E1 -13071.886,E2 -13071.886} C_VEL
LIN {X 0,Y 367.981,Z 299.612,A -85,B 0,C 180,E1 -13072.841,E2 -13072.841} C_VEL
LIN {X 0,Y 365.088,Z 286.226,A -85,B 0,C 180,E1 -13073.669,E2 -13073.669} C_VEL
LIN {X 0,Y 361.248,Z 272.067,A -85,B 0,C 180,E1 -13074.387,E2 -13074.387} C_VEL
LIN {X 0,Y 361.699,Z 266.718,A -85,B 0,C 180,E1 -13077.796,E2 -13077.796} C_VEL
LIN {X 0,Y 362.028,Z 262.86,A -85,B 0,C 180,E1 -13080.314,E2 -13080.314} C_VEL
LIN {X 0,Y 362.497,Z 257.073,A -85,B 0,C 180,E1 -13084.211,E2 -13084.211} C_VEL
LIN {X 0,Y 362.967,Z 252.376,A -85,B 0,C 180,E1 -13087.451,E2 -13087.451} C_VEL
LIN {X 0,Y 362.973,Z 249.26,A -85,B 0,C 180,E1 -13089.714,E2 -13089.714} C_VEL
LIN {X 0,Y 362.53,Z 245.374,A -85,B 0,C 180,E1 -13092.727,E2 -13092.727} C_VEL
LIN {X 0,Y 361.853,Z 241.064,A -85,B 0,C 180,E1 -13096.308,E2 -13096.308} C_VEL
LIN {X 0,Y 361.855,Z 241.038,A -85,B 0,C 180,E1 -13100.139,E2 -13100.139} C_VEL
LIN {X 0,Y 361.868,Z 241.038,A -85,B 0,C 180,E1 -13102.982,E2 -13102.982} C_VEL
LIN {X 0,Y 361.859,Z 241.037,A -85,B 0,C 180,E1 -13106.631,E2 -13106.631} C_VEL
LIN {X 0,Y 361.865,Z 241.035,A -85,B 0,C 180,E1 -13109.671,E2 -13109.671} C_VEL
LIN {X 0,Y 361.867,Z 241.034,A -85,B 0,C 180,E1 -13113.468,E2 -13113.468} C_VEL
LIN {X 0,Y 361.879,Z 241.035,A -85,B 0,C 180,E1 -13117.144,E2 -13117.144} C_VEL
LIN {X 0,Y 361.905,Z 241.031,A -85,B 0,C 180,E1 -13120.723,E2 -13120.723} C_VEL
LIN {X 0,Y 361.945,Z 241.024,A -85,B 0,C 180,E1 -13124.226,E2 -13124.226} C_VEL
LIN {X 0,Y 362,Z 241.015,A -85,B 0,C 180,E1 -13126.528,E2 -13126.528} C_VEL
LIN {X 0,Y 362.001,Z 241.013,A -85,B 0,C 180,E1 -13129.937,E2 -13129.937} C_VEL
LIN {X 0,Y 362.125,Z 241.003,A -85,B 0,C 180,E1 -13133.313,E2 -13133.313} C_VEL
LIN {X 0,Y 362.282,Z 240.982,A -85,B 0,C 180,E1 -13137.777,E2 -13137.777} C_VEL
LIN {X 0,Y 362.382,Z 240.972,A -85,B 0,C 180,E1 -13140,E2 -13140} C_VEL
LIN {X 0,Y 362.278,Z 240.982,A -85,B 0,C 180,E1 -13142.224,E2 -13142.224} C_VEL
LIN {X 0,Y 362.162,Z 240.998,A -85,B 0,C 180,E1 -13146.686,E2 -13146.686} C_VEL
LIN {X 0,Y 362.033,Z 241.014,A -85,B 0,C 180,E1 -13150.062,E2 -13150.062} C_VEL
LIN {X 0,Y 362,Z 241.016,A -85,B 0,C 180,E1 -13153.899,E2 -13153.899} C_VEL
LIN {X 0,Y 361.969,Z 241.023,A -85,B 0,C 180,E1 -13157.939,E2 -13157.939} C_VEL
LIN {X 0,Y 361.863,Z 241.034,A -85,B 0,C 180,E1 -13161.655,E2 -13161.655} C_VEL
LIN {X 0,Y 361.928,Z 241.026,A -85,B 0,C 180,E1 -13165.29,E2 -13165.29} C_VEL
LIN {X 0,Y 361.91,Z 241.03,A -85,B 0,C 180,E1 -13167.779,E2 -13167.779} C_VEL
LIN {X 0,Y 361.839,Z 241.037,A -85,B 0,C 180,E1 -13171.629,E2 -13171.629} C_VEL
LIN {X 0,Y 361.875,Z 241.035,A -85,B 0,C 180,E1 -13175.345,E2 -13175.345} C_VEL
LIN {X 0,Y 361.827,Z 241.041,A -85,B 0,C 180,E1 -13179.018,E2 -13179.018} C_VEL
LIN {X 0,Y 361.834,Z 241.041,A -85,B 0,C 180,E1 -13182.829,E2 -13182.829} C_VEL
LIN {X 0,Y 361.819,Z 241.042,A -85,B 0,C 180,E1 -13185.947,E2 -13185.947} C_VEL
LIN {X 0,Y 361.825,Z 241.222,A -85,B 0,C 180,E1 -13188.669,E2 -13188.669} C_VEL
LIN {X 0,Y 362.058,Z 244.179,A -85,B 0,C 180,E1 -13191.599,E2 -13191.599} C_VEL
LIN {X 0,Y 361.947,Z 247.444,A -85,B 0,C 180,E1 -13194.639,E2 -13194.639} C_VEL
LIN {X 0,Y 361.613,Z 251.612,A -85,B 0,C 180,E1 -13198.349,E2 -13198.349} C_VEL
LIN {X 0,Y 361.314,Z 256.128,A -85,B 0,C 180,E1 -13202.171,E2 -13202.171} C_VEL
LIN {X 0,Y 361.13,Z 260.459,A -85,B 0,C 180,E1 -13205.678,E2 -13205.678} C_VEL
LIN {X 0,Y 364.876,Z 272.564,A -85,B 0,C 180,E1 -13206.321,E2 -13206.321} C_VEL
LIN {X 0,Y 368.442,Z 285.942,A -85,B 0,C 180,E1 -13207.189,E2 -13207.189} C_VEL
LIN {X 0,Y 370.784,Z 297.872,A -85,B 0,C 180,E1 -13208.084,E2 -13208.084} C_VEL
LIN {X 0,Y 369.604,Z 311.543,A -85,B 0,C 180,E1 -13209.113,E2 -13209.113} C_VEL
LIN {X 0,Y 368.18,Z 324.407,A -85,B 0,C 180,E1 -13210.34,E2 -13210.34} C_VEL
LIN {X 0,Y 366.717,Z 335.982,A -85,B 0,C 180,E1 -13211.71,E2 -13211.71} C_VEL
LIN {X 0,Y 365.287,Z 346.457,A -85,B 0,C 180,E1 -13213.226,E2 -13213.226} C_VEL
LIN {X 0,Y 363.894,Z 356.202,A -85,B 0,C 180,E1 -13214.944,E2 -13214.944} C_VEL
LIN {X 0,Y 362.899,Z 364.916,A -85,B 0,C 180,E1 -13216.847,E2 -13216.847} C_VEL
LIN {X 0,Y 361.918,Z 372.173,A -85,B 0,C 180,E1 -13218.803,E2 -13218.803} C_VEL
LIN {X 0,Y 361.17,Z 378.688,A -85,B 0,C 180,E1 -13221.044,E2 -13221.044} C_VEL
LIN {X 0,Y 360.747,Z 383.571,A -85,B 0,C 180,E1 -13223.287,E2 -13223.287} C_VEL
LIN {X 0,Y 360.475,Z 386.969,A -85,B 0,C 180,E1 -13225.527,E2 -13225.527} C_VEL
LIN {X 0,Y 360.291,Z 388.988,A -85,B 0,C 180,E1 -13227.764,E2 -13227.764} C_VEL
LIN {X 0,Y 360.292,Z 389.679,A -85,B 0,C 180,E1 -13230,E2 -13230} C_VEL
LIN {X 0,Y 360.29,Z 389.054,A -85,B 0,C 180,E1 -13232.236,E2 -13232.236} C_VEL
LIN {X 0,Y 360.472,Z 387.095,A -85,B 0,C 180,E1 -13234.473,E2 -13234.473} C_VEL
LIN {X 0,Y 360.745,Z 383.758,A -85,B 0,C 180,E1 -13236.713,E2 -13236.713} C_VEL
LIN {X 0,Y 361.14,Z 378.944,A -85,B 0,C 180,E1 -13238.957,E2 -13238.957} C_VEL
LIN {X 0,Y 361.849,Z 372.497,A -85,B 0,C 180,E1 -13241.2,E2 -13241.2} C_VEL
LIN {X 0,Y 362.839,Z 365.313,A -85,B 0,C 180,E1 -13243.155,E2 -13243.155} C_VEL
LIN {X 0,Y 363.802,Z 356.979,A -85,B 0,C 180,E1 -13245.003,E2 -13245.003} C_VEL
LIN {X 0,Y 365.255,Z 347.086,A -85,B 0,C 180,E1 -13246.776,E2 -13246.776} C_VEL
LIN {X 0,Y 366.638,Z 336.739,A -85,B 0,C 180,E1 -13248.294,E2 -13248.294} C_VEL
LIN {X 0,Y 368.097,Z 325.317,A -85,B 0,C 180,E1 -13249.665,E2 -13249.665} C_VEL
LIN {X 0,Y 369.518,Z 312.654,A -85,B 0,C 180,E1 -13250.893,E2 -13250.893} C_VEL
LIN {X 0,Y 370.729,Z 299.72,A -85,B 0,C 180,E1 -13251.887,E2 -13251.887} C_VEL
LIN {X 0,Y 370.52,Z 296.024,A -85,B 0,C 180,E1 -13252.163,E2 -13252.163} C_VEL
LIN {X 0,Y 367.487,Z 282.071,A -85,B 0,C 180,E1 -13253.181,E2 -13253.181} C_VEL
LIN {X 0,Y 363.665,Z 268.573,A -85,B 0,C 180,E1 -13254.011,E2 -13254.011} C_VEL
LIN {X 0,Y 361.113,Z 260.335,A -85,B 0,C 180,E1 -13254.468,E2 -13254.468} C_VEL
LIN {X 0,Y 361.178,Z 258.598,A -85,B 0,C 180,E1 -13255.883,E2 -13255.883} C_VEL
LIN {X 0,Y 360.559,Z 257.566,A -85,B 0,C 180,E1 -13256.801,E2 -13256.801} C_VEL
LIN {X 0,Y 357.778,Z 256.118,A -85,B 0,C 180,E1 -13258.303,E2 -13258.303} C_VEL
LIN {X 0,Y 355.452,Z 254.977,A -85,B 0,C 180,E1 -13259.518,E2 -13259.518} C_VEL
LIN {X 0,Y 354.523,Z 254.011,A -85,B 0,C 180,E1 -13260.455,E2 -13260.455} C_VEL
LIN {X 0,Y 354.484,Z 253.656,A -85,B 0,C 180,E1 -13260.771,E2 -13260.771} C_VEL
LIN {X 0,Y 354.759,Z 250.356,A -85,B 0,C 180,E1 -13263.69,E2 -13263.69} C_VEL
LIN {X 0,Y 354.948,Z 247.377,A -85,B 0,C 180,E1 -13266.442,E2 -13266.442} C_VEL
LIN {X 0,Y 354.973,Z 244.262,A -85,B 0,C 180,E1 -13269.452,E2 -13269.452} C_VEL
LIN {X 0,Y 354.838,Z 242.569,A -85,B 0,C 180,E1 -13271.181,E2 -13271.181} C_VEL
LIN {X 0,Y 354.791,Z 241.918,A -85,B 0,C 180,E1 -13272.338,E2 -13272.338} C_VEL
LIN {X 0,Y 354.768,Z 241.924,A -85,B 0,C 180,E1 -13276.104,E2 -13276.104} C_VEL
LIN {X 0,Y 354.768,Z 241.921,A -85,B 0,C 180,E1 -13279.176,E2 -13279.176} C_VEL
LIN {X 0,Y 354.803,Z 241.915,A -85,B 0,C 180,E1 -13282.404,E2 -13282.404} C_VEL
LIN {X 0,Y 354.814,Z 241.913,A -85,B 0,C 180,E1 -13284.941,E2 -13284.941} C_VEL
LIN {X 0,Y 354.796,Z 241.915,A -85,B 0,C 180,E1 -13288.405,E2 -13288.405} C_VEL
LIN {X 0,Y 354.849,Z 241.908,A -85,B 0,C 180,E1 -13291.619,E2 -13291.619} C_VEL
LIN {X 0,Y 354.901,Z 241.901,A -85,B 0,C 180,E1 -13294.173,E2 -13294.173} C_VEL
LIN {X 0,Y 354.818,Z 241.912,A -85,B 0,C 180,E1 -13297.893,E2 -13297.893} C_VEL
LIN {X 0,Y 354.925,Z 241.9,A -85,B 0,C 180,E1 -13301.892,E2 -13301.892} C_VEL
LIN {X 0,Y 354.946,Z 241.896,A -85,B 0,C 180,E1 -13305.981,E2 -13305.981} C_VEL
LIN {X 0,Y 354.959,Z 241.893,A -85,B 0,C 180,E1 -13309.735,E2 -13309.735} C_VEL
LIN {X 0,Y 355.115,Z 241.876,A -85,B 0,C 180,E1 -13313.18,E2 -13313.18} C_VEL
LIN {X 0,Y 355.243,Z 241.858,A -85,B 0,C 180,E1 -13317.732,E2 -13317.732} C_VEL
LIN {X 0,Y 355.183,Z 241.867,A -85,B 0,C 180,E1 -13321.134,E2 -13321.134} C_VEL
LIN {X 0,Y 355.246,Z 241.857,A -85,B 0,C 180,E1 -13322.268,E2 -13322.268} C_VEL
LIN {X 0,Y 355.092,Z 241.878,A -85,B 0,C 180,E1 -13326.82,E2 -13326.82} C_VEL
LIN {X 0,Y 354.958,Z 241.895,A -85,B 0,C 180,E1 -13330.265,E2 -13330.265} C_VEL
LIN {X 0,Y 354.946,Z 241.897,A -85,B 0,C 180,E1 -13334.019,E2 -13334.019} C_VEL
LIN {X 0,Y 354.892,Z 241.905,A -85,B 0,C 180,E1 -13338.092,E2 -13338.092} C_VEL
LIN {X 0,Y 354.821,Z 241.914,A -85,B 0,C 180,E1 -13341.418,E2 -13341.418} C_VEL
LIN {X 0,Y 354.851,Z 241.907,A -85,B 0,C 180,E1 -13344.577,E2 -13344.577} C_VEL
LIN {X 0,Y 354.801,Z 241.914,A -85,B 0,C 180,E1 -13348.385,E2 -13348.385} C_VEL
LIN {X 0,Y 354.789,Z 241.918,A -85,B 0,C 180,E1 -13352.333,E2 -13352.333} C_VEL
LIN {X 0,Y 354.823,Z 241.917,A -85,B 0,C 180,E1 -13355.699,E2 -13355.699} C_VEL
LIN {X 0,Y 354.826,Z 241.914,A -85,B 0,C 180,E1 -13359.423,E2 -13359.423} C_VEL
LIN {X 0,Y 354.826,Z 241.978,A -85,B 0,C 180,E1 -13363.326,E2 -13363.326} C_VEL
LIN {X 0,Y 355.521,Z 246.3,A -85,B 0,C 180,E1 -13367.006,E2 -13367.006} C_VEL
LIN {X 0,Y 355.987,Z 250.522,A -85,B 0,C 180,E1 -13370.349,E2 -13370.349} C_VEL
LIN {X 0,Y 355.958,Z 253.1,A -85,B 0,C 180,E1 -13372.261,E2 -13372.261} C_VEL
LIN {X 0,Y 355.56,Z 256.988,A -85,B 0,C 180,E1 -13375.025,E2 -13375.025} C_VEL
LIN {X 0,Y 355.149,Z 261.727,A -85,B 0,C 180,E1 -13378.312,E2 -13378.312} C_VEL
LIN {X 0,Y 354.711,Z 266.606,A -85,B 0,C 180,E1 -13381.607,E2 -13381.607} C_VEL
LIN {X 0,Y 354.257,Z 272.066,A -85,B 0,C 180,E1 -13385.093,E2 -13385.093} C_VEL
LIN {X 0,Y 358.186,Z 286.2,A -85,B 0,C 180,E1 -13385.835,E2 -13385.835} C_VEL
LIN {X 0,Y 361.047,Z 299.077,A -85,B 0,C 180,E1 -13386.656,E2 -13386.656} C_VEL
LIN {X 0,Y 362.94,Z 310.635,A -85,B 0,C 180,E1 -13387.515,E2 -13387.515} C_VEL
LIN {X 0,Y 363.332,Z 316.59,A -85,B 0,C 180,E1 -13387.989,E2 -13387.989} C_VEL
LIN {X 0,Y 361.91,Z 329.712,A -85,B 0,C 180,E1 -13389.091,E2 -13389.091} C_VEL
LIN {X 0,Y 360.35,Z 341.64,A -85,B 0,C 180,E1 -13390.34,E2 -13390.34} C_VEL
LIN {X 0,Y 358.892,Z 352.513,A -85,B 0,C 180,E1 -13391.74,E2 -13391.74} C_VEL
LIN {X 0,Y 357.378,Z 363.259,A -85,B 0,C 180,E1 -13393.432,E2 -13393.432} C_VEL
LIN {X 0,Y 356.141,Z 372.573,A -85,B 0,C 180,E1 -13395.229,E2 -13395.229} C_VEL
LIN {X 0,Y 355.156,Z 380.645,A -85,B 0,C 180,E1 -13397.137,E2 -13397.137} C_VEL
LIN {X 0,Y 354.234,Z 387.501,A -85,B 0,C 180,E1 -13399.136,E2 -13399.136} C_VEL
LIN {X 0,Y 353.779,Z 392.23,A -85,B 0,C 180,E1 -13400.855,E2 -13400.855} C_VEL
LIN {X 0,Y 353.412,Z 397.131,A -85,B 0,C 180,E1 -13403.147,E2 -13403.147} C_VEL
LIN {X 0,Y 353.243,Z 400.539,A -85,B 0,C 180,E1 -13405.435,E2 -13405.435} C_VEL
LIN {X 0,Y 353.141,Z 402.554,A -85,B 0,C 180,E1 -13407.719,E2 -13407.719} C_VEL
LIN {X 0,Y 353.191,Z 403.221,A -85,B 0,C 180,E1 -13410,E2 -13410} C_VEL
LIN {X 0,Y 353.141,Z 402.548,A -85,B 0,C 180,E1 -13412.281,E2 -13412.281} C_VEL
LIN {X 0,Y 353.24,Z 400.528,A -85,B 0,C 180,E1 -13414.565,E2 -13414.565} C_VEL
LIN {X 0,Y 353.412,Z 397.112,A -85,B 0,C 180,E1 -13416.853,E2 -13416.853} C_VEL
LIN {X 0,Y 353.764,Z 392.198,A -85,B 0,C 180,E1 -13419.145,E2 -13419.145} C_VEL
LIN {X 0,Y 354.417,Z 385.644,A -85,B 0,C 180,E1 -13421.437,E2 -13421.437} C_VEL
LIN {X 0,Y 355.387,Z 378.356,A -85,B 0,C 180,E1 -13423.436,E2 -13423.436} C_VEL
LIN {X 0,Y 356.361,Z 370.717,A -85,B 0,C 180,E1 -13425.148,E2 -13425.148} C_VEL
LIN {X 0,Y 357.597,Z 361.555,A -85,B 0,C 180,E1 -13426.851,E2 -13426.851} C_VEL
LIN {X 0,Y 359.123,Z 350.446,A -85,B 0,C 180,E1 -13428.543,E2 -13428.543} C_VEL
LIN {X 0,Y 360.705,Z 339.108,A -85,B 0,C 180,E1 -13429.936,E2 -13429.936} C_VEL
LIN {X 0,Y 362.194,Z 327.439,A -85,B 0,C 180,E1 -13431.104,E2 -13431.104} C_VEL
LIN {X 0,Y 363.382,Z 314.439,A -85,B 0,C 180,E1 -13432.157,E2 -13432.157} C_VEL
LIN {X 0,Y 361.567,Z 302.117,A -85,B 0,C 180,E1 -13433.116,E2 -13433.116} C_VEL
LIN {X 0,Y 358.59,Z 287.842,A -85,B 0,C 180,E1 -13434.051,E2 -13434.051} C_VEL
LIN {X 0,Y 354.709,Z 274.148,A -85,B 0,C 180,E1 -13434.803,E2 -13434.803} C_VEL
LIN {X 0,Y 354.256,Z 271.929,A -85,B 0,C 180,E1 -13434.903,E2 -13434.903} C_VEL
LIN {X 0,Y 354.71,Z 266.58,A -85,B 0,C 180,E1 -13438.393,E2 -13438.393} C_VEL
LIN {X 0,Y 355.138,Z 261.704,A -85,B 0,C 180,E1 -13441.685,E2 -13441.685} C_VEL
LIN {X 0,Y 355.55,Z 256.956,A -85,B 0,C 180,E1 -13444.976,E2 -13444.976} C_VEL
LIN {X 0,Y 355.958,Z 252.917,A -85,B 0,C 180,E1 -13447.837,E2 -13447.837} C_VEL
LIN {X 0,Y 355.873,Z 249.151,A -85,B 0,C 180,E1 -13450.67,E2 -13450.67} C_VEL
LIN {X 0,Y 355.351,Z 245.268,A -85,B 0,C 180,E1 -13453.806,E2 -13453.806} C_VEL
LIN {X 0,Y 354.792,Z 241.919,A -85,B 0,C 180,E1 -13456.808,E2 -13456.808} C_VEL
LIN {X 0,Y 354.816,Z 241.916,A -85,B 0,C 180,E1 -13460.666,E2 -13460.666} C_VEL
LIN {X 0,Y 354.822,Z 241.917,A -85,B 0,C 180,E1 -13464.301,E2 -13464.301} C_VEL
LIN {X 0,Y 354.788,Z 241.92,A -85,B 0,C 180,E1 -13467.667,E2 -13467.667} C_VEL
LIN {X 0,Y 354.802,Z 241.914,A -85,B 0,C 180,E1 -13471.615,E2 -13471.615} C_VEL
LIN {X 0,Y 354.835,Z 241.913,A -85,B 0,C 180,E1 -13475.657,E2 -13475.657} C_VEL
LIN {X 0,Y 354.828,Z 241.913,A -85,B 0,C 180,E1 -13479.113,E2 -13479.113} C_VEL
LIN {X 0,Y 354.881,Z 241.903,A -85,B 0,C 180,E1 -13482.719,E2 -13482.719} C_VEL
LIN {X 0,Y 354.953,Z 241.892,A -85,B 0,C 180,E1 -13486.255,E2 -13486.255} C_VEL
LIN {X 0,Y 354.957,Z 241.889,A -85,B 0,C 180,E1 -13489.735,E2 -13489.735} C_VEL
LIN {X 0,Y 355.09,Z 241.878,A -85,B 0,C 180,E1 -13493.18,E2 -13493.18} C_VEL
LIN {X 0,Y 355.245,Z 241.858,A -85,B 0,C 180,E1 -13497.732,E2 -13497.732} C_VEL
LIN {X 0,Y 355.333,Z 241.85,A -85,B 0,C 180,E1 -13500,E2 -13500} C_VEL
LIN {X 0,Y 355.241,Z 241.859,A -85,B 0,C 180,E1 -13502.268,E2 -13502.268} C_VEL
LIN {X 0,Y 355.126,Z 241.874,A -85,B 0,C 180,E1 -13506.82,E2 -13506.82} C_VEL
LIN {X 0,Y 354.98,Z 241.892,A -85,B 0,C 180,E1 -13510.264,E2 -13510.264} C_VEL
LIN {X 0,Y 354.944,Z 241.895,A -85,B 0,C 180,E1 -13514.019,E2 -13514.019} C_VEL
LIN {X 0,Y 354.925,Z 241.9,A -85,B 0,C 180,E1 -13518.109,E2 -13518.109} C_VEL
LIN {X 0,Y 354.817,Z 241.911,A -85,B 0,C 180,E1 -13522.107,E2 -13522.107} C_VEL
LIN {X 0,Y 354.9,Z 241.903,A -85,B 0,C 180,E1 -13525.828,E2 -13525.828} C_VEL
LIN {X 0,Y 354.819,Z 241.912,A -85,B 0,C 180,E1 -13529.682,E2 -13529.682} C_VEL
LIN {X 0,Y 354.807,Z 241.915,A -85,B 0,C 180,E1 -13533.702,E2 -13533.702} C_VEL
LIN {X 0,Y 354.797,Z 241.915,A -85,B 0,C 180,E1 -13536.46,E2 -13536.46} C_VEL
LIN {X 0,Y 354.769,Z 241.918,A -85,B 0,C 180,E1 -13539.413,E2 -13539.413} C_VEL
LIN {X 0,Y 354.786,Z 241.919,A -85,B 0,C 180,E1 -13542.867,E2 -13542.867} C_VEL
LIN {X 0,Y 354.768,Z 241.92,A -85,B 0,C 180,E1 -13546.104,E2 -13546.104} C_VEL
LIN {X 0,Y 354.792,Z 241.919,A -85,B 0,C 180,E1 -13547.662,E2 -13547.662} C_VEL
LIN {X 0,Y 354.902,Z 242.815,A -85,B 0,C 180,E1 -13549.195,E2 -13549.195} C_VEL
LIN {X 0,Y 355.022,Z 245.992,A -85,B 0,C 180,E1 -13552.358,E2 -13552.358} C_VEL
LIN {X 0,Y 354.861,Z 248.747,A -85,B 0,C 180,E1 -13554.946,E2 -13554.946} C_VEL
LIN {X 0,Y 354.564,Z 252.655,A -85,B 0,C 180,E1 -13558.466,E2 -13558.466} C_VEL
LIN {X 0,Y 354.277,Z 256.253,A -85,B 0,C 180,E1 -13561.569,E2 -13561.569} C_VEL
LIN {X 0,Y 354.08,Z 260.509,A -85,B 0,C 180,E1 -13565.154,E2 -13565.154} C_VEL
LIN {X 0,Y 357,Z 269.849,A -85,B 0,C 180,E1 -13565.658,E2 -13565.658} C_VEL
LIN {X 0,Y 360.669,Z 282.726,A -85,B 0,C 180,E1 -13566.487,E2 -13566.487} C_VEL
LIN {X 0,Y 363.29,Z 294.554,A -85,B 0,C 180,E1 -13567.37,E2 -13567.37} C_VEL
LIN {X 0,Y 364.082,Z 300.124,A -85,B 0,C 180,E1 -13567.818,E2 -13567.818} C_VEL
LIN {X 0,Y 362.812,Z 313.262,A -85,B 0,C 180,E1 -13568.852,E2 -13568.852} C_VEL
LIN {X 0,Y 361.34,Z 325.835,A -85,B 0,C 180,E1 -13570.1,E2 -13570.1} C_VEL
